# B&R Automation Studio project NAINV104C00R8L515F00 (part 8)

#### fHermesIllegalMsgNotAvlNotRdyDS.st
```iecst
(* Hermes Illegal Message - Not Available Not Ready For Downstream *)
FUNCTION fHermesIllegalMsgNotAvlNotRdyDS

	IF tyMsgType.bServiceDescription = TRUE THEN

		fHermesIllegalMsgNotAvlNotRdyDS	:= 2857;	//Receive ServiceDescription While Downstream In Not Available Not Ready State

	ELSIF tyMsgType.bBoardAvailable = TRUE THEN

		fHermesIllegalMsgNotAvlNotRdyDS	:= 2858;	//Receive BoardAvailable While Downstream In Not Available Not Ready State

	ELSIF tyMsgType.bRevokeBoardAvailable = TRUE THEN

		fHermesIllegalMsgNotAvlNotRdyDS	:= 2859;	//Receive RevokeBoardAvailable While Downstream In Not Available Not Ready State

	ELSIF tyMsgType.bRevokeMachineReady = TRUE THEN

		fHermesIllegalMsgNotAvlNotRdyDS	:= 2860;	//Receive RevokeMachineReady While Downstream In Not Available Not Ready State

	ELSIF tyMsgType.bStartTransport = TRUE THEN

		fHermesIllegalMsgNotAvlNotRdyDS	:= 2861;	//Receive StartTransport While Downstream In Not Available Not Ready State

	ELSIF tyMsgType.bStopTransport = TRUE THEN

		fHermesIllegalMsgNotAvlNotRdyDS	:= 2862;	//Receive StopTransport While Downstream In Not Available Not Ready State

	ELSIF tyMsgType.bTransportFinished = TRUE THEN

		fHermesIllegalMsgNotAvlNotRdyDS	:= 2863;	//Receive TransportFinished While Downstream In Not Available Not Ready State

	ELSIF tyMsgType.bBoardForecast = TRUE THEN

		fHermesIllegalMsgNotAvlNotRdyDS	:= 2864;	//Receive BoardForecast While Downstream In Not Available Not Ready State

	ELSE

		fHermesIllegalMsgNotAvlNotRdyDS	:= 0;

	END_IF

END_FUNCTION
```

#### fHermesIllegalMsgBrdAvlDS.st
```iecst
(* Hermes Illegal Message - Board Available For Downstream *)
FUNCTION fHermesIllegalMsgBrdAvlDS

	IF tyMsgType.bServiceDescription = TRUE THEN

		fHermesIllegalMsgBrdAvlDS	:= 2865;	//Receive ServiceDescription While Downstream In Board Available State

	ELSIF tyMsgType.bBoardAvailable = TRUE THEN

		fHermesIllegalMsgBrdAvlDS	:= 2866;	//Receive BoardAvailable While Downstream In Board Available State

	ELSIF tyMsgType.bRevokeBoardAvailable = TRUE THEN

		fHermesIllegalMsgBrdAvlDS	:= 2867;	//Receive RevokeBoardAvailable While Downstream In Board Available State

	ELSIF tyMsgType.bRevokeMachineReady = TRUE THEN

		fHermesIllegalMsgBrdAvlDS	:= 2868;	//Receive RevokeMachineReady While Downstream In Board Available State

	ELSIF (tyMsgType.bStartTransport = TRUE) AND (tyMsgType.bMachineReady = FALSE) THEN	//To Take Care When Machine Ready And StartTransport Receive In One Message

		fHermesIllegalMsgBrdAvlDS	:= 2869;	//Receive StartTransport While Downstream In Board Available State

	ELSIF tyMsgType.bStopTransport = TRUE THEN

		fHermesIllegalMsgBrdAvlDS	:= 2870;	//Receive StopTransport While Downstream In Board Available State

	ELSIF tyMsgType.bTransportFinished = TRUE THEN

		fHermesIllegalMsgBrdAvlDS	:= 2871;	//Receive TransportFinished While Downstream In Board Available State

	ELSIF tyMsgType.bBoardForecast = TRUE THEN

		fHermesIllegalMsgBrdAvlDS	:= 2872;	//Receive BoardForecast While Downstream In Board Available State

	ELSE

		fHermesIllegalMsgBrdAvlDS	:= 0;

	END_IF

END_FUNCTION
```

#### fHermesIllegalMsgMcRdyDS.st
```iecst
(* Hermes Illegal Message - Machine Ready For Downstream *)
FUNCTION fHermesIllegalMsgMcRdyDS

	IF tyMsgType.bServiceDescription = TRUE THEN

		fHermesIllegalMsgMcRdyDS	:= 2873;	//Receive ServiceDescription While Downstream In Machine Ready State

	ELSIF tyMsgType.bBoardAvailable = TRUE THEN

		fHermesIllegalMsgMcRdyDS	:= 2874;	//Receive BoardAvailable While Downstream In Machine Ready State

	ELSIF tyMsgType.bRevokeBoardAvailable = TRUE THEN

		fHermesIllegalMsgMcRdyDS	:= 2875;	//Receive RevokeBoardAvailable While Downstream In Machine Ready State

	ELSIF tyMsgType.bMachineReady = TRUE THEN

		fHermesIllegalMsgMcRdyDS	:= 2876;	//Receive MachineReady While Downstream In Machine Ready State

	ELSIF tyMsgType.bStopTransport = TRUE THEN

		fHermesIllegalMsgMcRdyDS	:= 2877;	//Receive StopTransport While Downstream In Machine Ready State

	ELSIF tyMsgType.bTransportFinished = TRUE THEN

		fHermesIllegalMsgMcRdyDS	:= 2878;	//Receive TransportFinished While Downstream In Machine Ready State

	ELSIF tyMsgType.bBoardForecast = TRUE THEN

		fHermesIllegalMsgMcRdyDS	:= 2879;	//Receive BoardForecast While Downstream In Machine Ready State

	ELSE

		fHermesIllegalMsgMcRdyDS	:= 0;

	END_IF

END_FUNCTION
```

#### fHermesIllegalMsgAvlAndRdyDS.st
```iecst
(* Hermes Illegal Message - Available And Ready For Downstream *)
FUNCTION fHermesIllegalMsgAvlAndRdyDS

	IF tyMsgType.bServiceDescription = TRUE THEN

		fHermesIllegalMsgAvlAndRdyDS	:= 2880;	//Receive ServiceDescription While Downstream In Available And Ready State

	ELSIF tyMsgType.bBoardAvailable = TRUE THEN

		fHermesIllegalMsgAvlAndRdyDS	:= 2881;	//Receive BoardAvailable While Downstream In Available And Ready State

	ELSIF tyMsgType.bRevokeBoardAvailable = TRUE THEN

		fHermesIllegalMsgAvlAndRdyDS	:= 2882;	//Receive RevokeBoardAvailable While Downstream In Available And Ready State

	ELSIF tyMsgType.bMachineReady = TRUE THEN

		fHermesIllegalMsgAvlAndRdyDS	:= 2883;	//Receive MachineReady While Downstream In Available And Ready State

	ELSIF tyMsgType.bStopTransport = TRUE THEN

		fHermesIllegalMsgAvlAndRdyDS	:= 2884;	//Receive StopTransport While Downstream In Available And Ready State

	ELSIF tyMsgType.bTransportFinished = TRUE THEN

		fHermesIllegalMsgAvlAndRdyDS	:= 2885;	//Receive TransportFinished While Downstream In Available And Ready State

	ELSIF tyMsgType.bBoardForecast = TRUE THEN

		fHermesIllegalMsgAvlAndRdyDS	:= 2886;	//Receive BoardForecast While Downstream In Available And Ready State

	ELSE

		fHermesIllegalMsgAvlAndRdyDS	:= 0;

	END_IF

END_FUNCTION
```

#### fHermesIllegalMsgTransportingDS.st
```iecst
(* Hermes Illegal Message - Transporting For Downstream *)
FUNCTION fHermesIllegalMsgTransportingDS

	IF tyMsgType.bServiceDescription = TRUE THEN

		fHermesIllegalMsgTransportingDS	:= 2887;	//Receive ServiceDescription While Downstream In Transporting State

	ELSIF tyMsgType.bBoardAvailable = TRUE THEN

		fHermesIllegalMsgTransportingDS	:= 2888;	//Receive BoardAvailable While Downstream In Transporting State

	ELSIF tyMsgType.bRevokeBoardAvailable = TRUE THEN

		fHermesIllegalMsgTransportingDS	:= 2889;	//Receive RevokeBoardAvailable While Downstream In Transporting State

	ELSIF tyMsgType.bMachineReady = TRUE THEN

		fHermesIllegalMsgTransportingDS	:= 2890;	//Receive MachineReady While Downstream In Transporting State

	ELSIF tyMsgType.bRevokeMachineReady = TRUE THEN

		fHermesIllegalMsgTransportingDS	:= 2891;	//Receive RevokeMachineReady While Downstream In Transporting State

	ELSIF tyMsgType.bStartTransport = TRUE THEN

		fHermesIllegalMsgTransportingDS	:= 2892;	//Receive StartTransport While Downstream In Transporting State

	ELSIF tyMsgType.bTransportFinished = TRUE THEN

		fHermesIllegalMsgTransportingDS	:= 2893;	//Receive TransportFinished While Downstream In Transporting State

	ELSIF tyMsgType.bBoardForecast = TRUE THEN

		fHermesIllegalMsgTransportingDS	:= 2894;	//Receive BoardForecast While Downstream In Transporting State

	ELSE

		fHermesIllegalMsgTransportingDS	:= 0;

	END_IF

END_FUNCTION
```

#### fHermesIllegalMsgTransportFiniDS.st
```iecst
(* Hermes Illegal Message - Transport Finished For Downstream *)
FUNCTION fHermesIllegalMsgTransportFiniDS

	IF tyMsgType.bServiceDescription = TRUE THEN

		fHermesIllegalMsgTransportFiniDS	:= 2895;	//Receive ServiceDescription While In Transport Finished State

	ELSIF tyMsgType.bBoardAvailable = TRUE THEN

		fHermesIllegalMsgTransportFiniDS	:= 2896;	//Receive BoardAvailable While In Transport Finished State

	ELSIF tyMsgType.bRevokeBoardAvailable = TRUE THEN

		fHermesIllegalMsgTransportFiniDS	:= 2897;	//Receive RevokeBoardAvailable While In Transport Finished State

	ELSIF tyMsgType.bMachineReady = TRUE THEN

		fHermesIllegalMsgTransportFiniDS	:= 2898;	//Receive MachineReady While In Transport Finished State

	ELSIF tyMsgType.bRevokeMachineReady = TRUE THEN

		fHermesIllegalMsgTransportFiniDS	:= 2899;	//Receive RevokeMachineReady While In Transport Finished State

	ELSIF tyMsgType.bStartTransport = TRUE THEN

		fHermesIllegalMsgTransportFiniDS	:= 2900;	//Receive StartTransport While In Transport Finished State

	ELSIF tyMsgType.bTransportFinished = TRUE THEN

		fHermesIllegalMsgTransportFiniDS	:= 2901;	//Receive TransportFinished While In Transport Finished State

	ELSIF tyMsgType.bBoardForecast = TRUE THEN

		fHermesIllegalMsgTransportFiniDS	:= 2902;	//Receive BoardForecast While In Transport Finished State

	ELSE

		fHermesIllegalMsgTransportFiniDS	:= 0;

	END_IF

END_FUNCTION
```

#### fHermesIllegalMsgTransportStopDS.st
```iecst
(* Hermes Illegal Message - Transport Stopped For Downstream *)
FUNCTION fHermesIllegalMsgTransportStopDS

	IF tyMsgType.bServiceDescription = TRUE THEN

		fHermesIllegalMsgTransportStopDS	:= 2903;	//Receive ServiceDescription While Downstream In Transport Stopped State

	ELSIF tyMsgType.bBoardAvailable = TRUE THEN

		fHermesIllegalMsgTransportStopDS	:= 2904;	//Receive BoardAvailable While Downstream In Transport Stopped State

	ELSIF tyMsgType.bRevokeBoardAvailable = TRUE THEN

		fHermesIllegalMsgTransportStopDS	:= 2905;	//Receive RevokeBoardAvailable While Downstream In Transport Stopped State

	ELSIF tyMsgType.bMachineReady = TRUE THEN

		fHermesIllegalMsgTransportStopDS	:= 2906;	//Receive MachineReady While Downstream In Transport Stopped State

	ELSIF tyMsgType.bRevokeMachineReady = TRUE THEN

		fHermesIllegalMsgTransportStopDS	:= 2907;	//Receive RevokeMachineReady While Downstream In Transport Stopped State

	ELSIF tyMsgType.bStartTransport = TRUE THEN

		fHermesIllegalMsgTransportStopDS	:= 2908;	//Receive StartTransport While Downstream In Transport Stopped State

	ELSIF tyMsgType.bStopTransport = TRUE THEN

		fHermesIllegalMsgTransportStopDS	:= 2909;	//Receive StopTransport While Downstream In Transport Stopped State

	ELSIF tyMsgType.bTransportFinished = TRUE THEN

		fHermesIllegalMsgTransportStopDS	:= 2910;	//Receive TransportFinished While Downstream In Transport Stopped State

	ELSIF tyMsgType.bBoardForecast = TRUE THEN

		fHermesIllegalMsgTransportStopDS	:= 2911;	//Receive BoardForecast While Downstream In Transport Stopped State

	ELSE

		fHermesIllegalMsgTransportStopDS	:= 0;

	END_IF

END_FUNCTION
```

#### fHermesIllegalMsgNotConnectedSvy.st
```iecst
(* Hermes Illegal Message - Not Connected For Supervisory *)
FUNCTION fHermesIllegalMsgNotConnectedSvy

	IF tyMsgType.bSetConfiguration = TRUE THEN

		fHermesIllegalMsgNotConnectedSvy	:= 2940;	//Receive SetConfiguration While Supervisory In Not Connected State

	ELSIF tyMsgType.bGetConfiguration = TRUE THEN

		fHermesIllegalMsgNotConnectedSvy	:= 2941;	//Receive GetConfiguration While Supervisory In Not Connected State

	ELSIF tyMsgType.bCurrentConfiguration = TRUE THEN

		fHermesIllegalMsgNotConnectedSvy	:= 2942;	//Receive CurrConfiguration While Supervisory In Not Connected State

	ELSIF tyMsgType.bSendWorkOrderInfo = TRUE THEN

		fHermesIllegalMsgNotConnectedSvy	:= 2943;	//Receive SendWorkOrderInfo While Supervisory In Not Connected State

	ELSIF tyMsgType.bQueryWorkOrderInfo = TRUE THEN

		fHermesIllegalMsgNotConnectedSvy	:= 2944;	//Receive QueryWorkOrderInfo While Supervisory In Not Connected State

	ELSIF tyMsgType.bBoardArrived = TRUE THEN

		fHermesIllegalMsgNotConnectedSvy	:= 2945;	//Receive BoardArrived While Supervisory In Not Connected State

	ELSIF tyMsgType.bBoardDeparted = TRUE THEN

		fHermesIllegalMsgNotConnectedSvy	:= 2946;	//Receive BoardDeparted While Supervisory In Not Connected State

	ELSE

		fHermesIllegalMsgNotConnectedSvy	:= 0;

	END_IF

END_FUNCTION
```

#### fHermesIllegalMsgSrvcDescripSvy.st
```iecst
(* Hermes Illegal Message - Supervisory Service Description *)
FUNCTION fHermesIllegalMsgSrvcDescripSvy

	IF tyMsgType.bSServiceDescription = TRUE THEN

		fHermesIllegalMsgSrvcDescripSvy	:= 2951;	//Receive Supervisory ServiceDescription While Supervisory In Service Description State

	ELSIF tyMsgType.bSetConfiguration = TRUE THEN

		fHermesIllegalMsgSrvcDescripSvy	:= 2952;	//Receive SetConfiguration While Supervisory In Service Description State

	ELSIF tyMsgType.bGetConfiguration = TRUE THEN

		fHermesIllegalMsgSrvcDescripSvy	:= 2953;	//Receive GetConfiguration While Supervisory In Service Description State

	ELSIF tyMsgType.bCurrentConfiguration = TRUE THEN

		fHermesIllegalMsgSrvcDescripSvy	:= 2954;	//Receive CurrConfiguration While Supervisory In Service Description State

	ELSIF tyMsgType.bSendWorkOrderInfo = TRUE THEN

		fHermesIllegalMsgSrvcDescripSvy	:= 2955;	//Receive SendWorkOrderInfo While Supervisory In Service Description State

	ELSIF tyMsgType.bQueryWorkOrderInfo = TRUE THEN

		fHermesIllegalMsgSrvcDescripSvy	:= 2956;	//Receive QueryWorkOrderInfo While Supervisory In Service Description State

	ELSIF tyMsgType.bBoardArrived = TRUE THEN

		fHermesIllegalMsgSrvcDescripSvy	:= 2957;	//Receive BoardArrived While Supervisory In Service Description State

	ELSIF tyMsgType.bBoardDeparted = TRUE THEN

		fHermesIllegalMsgSrvcDescripSvy	:= 2958;	//Receive BoardDeparted While Supervisory In Service Description State

	ELSE

		fHermesIllegalMsgSrvcDescripSvy	:= 0;

	END_IF

END_FUNCTION
```

#### fHermesIllegalMsgConnectedSvy.st
```iecst
(* Hermes Illegal Message - Connected For Supervisory *)
FUNCTION fHermesIllegalMsgConnectedSvy

	IF tyMsgType.bServiceDescription = TRUE THEN

		fHermesIllegalMsgConnectedSvy	:= 2963;	//Receive Supervisory ServiceDescription While Supervisory In Connected State

	ELSIF tyMsgType.bCurrentConfiguration = TRUE THEN

		fHermesIllegalMsgConnectedSvy	:= 2964;	//Receive CurrConfiguration While Supervisory In Connected State

	ELSIF tyMsgType.bQueryWorkOrderInfo = TRUE THEN

		fHermesIllegalMsgConnectedSvy	:= 2965;	//Receive QueryWorkOrderInfo While Supervisory In Connected State

	ELSIF tyMsgType.bBoardArrived = TRUE THEN

		fHermesIllegalMsgConnectedSvy	:= 2966;	//Receive BoardArrived While Supervisory In Connected State

	ELSIF tyMsgType.bBoardDeparted = TRUE THEN

		fHermesIllegalMsgConnectedSvy	:= 2967;	//Receive BoardDeparted While Supervisory In Connected State

	ELSE

		fHermesIllegalMsgConnectedSvy	:= 0;

	END_IF

END_FUNCTION
```

#### fHermesGenerateUUID.st
```iecst
(* Hermes Generate UUID *)
FUNCTION fHermesGenerateUUID

	fHermesGenerateUUID	:= TRUE;

	memset(ADR(p_sUUID) , 0 , SIZEOF(p_sUUID));

	//Year Difference: From 1970
	fConvertUSINTToHex(ADR(sTemp2) , UINT_TO_USINT((tyDTStructure.year - 1970)));
	p_sUUID	:= sTemp2;

	//Month
	fConvertUSINTToHex(ADR(sTemp2) , tyDTStructure.month);
	memcpy(ADR(p_sUUID) + LEN(p_sUUID) , ADR(sTemp2) , 2);

	//Day
	fConvertUSINTToHex(ADR(sTemp2) , tyDTStructure.day);
	memcpy(ADR(p_sUUID) + LEN(p_sUUID) , ADR(sTemp2) , 2);

	//Hour
	fConvertUSINTToHex(ADR(sTemp2) , tyDTStructure.hour);
	memcpy(ADR(p_sUUID) + LEN(p_sUUID) , ADR(sTemp2) , 2);
	memcpy(ADR(p_sUUID) + LEN(p_sUUID) , ADR('-') , 1);

	//Minute
	fConvertUSINTToHex(ADR(sTemp2) , tyDTStructure.minute);
	memcpy(ADR(p_sUUID) + LEN(p_sUUID) , ADR(sTemp2) , 2);

	//Second
	fConvertUSINTToHex(ADR(sTemp2) , tyDTStructure.second);
	memcpy(ADR(p_sUUID) + LEN(p_sUUID) , ADR(sTemp2) , 2);
	memcpy(ADR(p_sUUID) + LEN(p_sUUID) , ADR('-') , 1);

	//Millisec
	fConvertUINTToHex(ADR(sTemp4) , tyDTStructure.millisec);
	memcpy(ADR(p_sUUID) + LEN(p_sUUID) , ADR(sTemp4) , 4);
	memcpy(ADR(p_sUUID) + LEN(p_sUUID) , ADR('-') , 1);

	//Microsec
	fConvertUINTToHex(ADR(sTemp4) , tyDTStructure.microsec);
	memcpy(ADR(p_sUUID) + LEN(p_sUUID) , ADR(sTemp4) , 4);
	memcpy(ADR(p_sUUID) + LEN(p_sUUID) , ADR('-') , 1);

	//Mac Address
	fConvertUSINTToHex(ADR(sTemp2) , a_usiMacAddr[0]);
	memcpy(ADR(p_sUUID) + LEN(p_sUUID) , ADR(sTemp2) , 2);

	fConvertUSINTToHex(ADR(sTemp2) , a_usiMacAddr[1]);
	memcpy(ADR(p_sUUID) + LEN(p_sUUID) , ADR(sTemp2) , 2);

	fConvertUSINTToHex(ADR(sTemp2) , a_usiMacAddr[2]);
	memcpy(ADR(p_sUUID) + LEN(p_sUUID) , ADR(sTemp2) , 2);

	fConvertUSINTToHex(ADR(sTemp2) , a_usiMacAddr[3]);
	memcpy(ADR(p_sUUID) + LEN(p_sUUID) , ADR(sTemp2) , 2);

	fConvertUSINTToHex(ADR(sTemp2) , a_usiMacAddr[4]);
	memcpy(ADR(p_sUUID) + LEN(p_sUUID) , ADR(sTemp2) , 2);

	fConvertUSINTToHex(ADR(sTemp2) , a_usiMacAddr[5]);
	memcpy(ADR(p_sUUID) + LEN(p_sUUID) , ADR(sTemp2) , 2);

END_FUNCTION
```

#### fHermesGetTimestamp.st
```iecst
(* Hermes Get Timestamp *)
FUNCTION fHermesGetTimestamp

	fHermesGetTimestamp	:= TRUE;

	memset(ADR(p_sTimestamp) , 0 , SIZEOF(p_sTimestamp));
	memset(ADR(sYear) , 0 , SIZEOF(sYear));
	memset(ADR(sMonth) , 0 , SIZEOF(sMonth));
	memset(ADR(sDay) , 0 , SIZEOF(sDay));
	memset(ADR(sHour) , 0 , SIZEOF(sHour));
	memset(ADR(sMinute) , 0 , SIZEOF(sMinute));
	memset(ADR(sSecond) , 0 , SIZEOF(sSecond));
	memset(ADR(sMillisec) , 0 , SIZEOF(sMillisec));

	sYear	:= UINT_TO_STRING(tyDTStructure.year);

	IF tyDTStructure.year < 10 THEN
		memcpy(ADR(sYear) + 3 , ADR(sYear) , 1);
		memcpy(ADR(sYear) , ADR('000') , 3);
	ELSIF tyDTStructure.year < 100 THEN
		memcpy(ADR(sYear) + 2 , ADR(sYear) , 2);
		memcpy(ADR(sYear) , ADR('000') , 2);
	ELSIF tyDTStructure.year < 1000 THEN
		memcpy(ADR(sYear) + 1 , ADR(sYear) , 3);
		memcpy(ADR(sYear) , ADR('000') , 1);
	END_IF

	sMonth	:= USINT_TO_STRING(tyDTStructure.month);

	IF tyDTStructure.month < 10 THEN
		memcpy(ADR(sMonth) + 1 , ADR(sMonth) , 1);
		memcpy(ADR(sMonth) , ADR('0') , 1);
	END_IF

	sDay	:= USINT_TO_STRING(tyDTStructure.day);

	IF tyDTStructure.day < 10 THEN
		memcpy(ADR(sDay) + 1 , ADR(sDay) , 1);
		memcpy(ADR(sDay) , ADR('0') , 1);
	END_IF

	sHour	:= USINT_TO_STRING(tyDTStructure.hour);

	IF tyDTStructure.hour < 10 THEN
		memcpy(ADR(sHour) + 1 , ADR(sHour) , 1);
		memcpy(ADR(sHour) , ADR('0') , 1);
	END_IF

	sMinute	:= USINT_TO_STRING(tyDTStructure.minute);

	IF tyDTStructure.minute < 10 THEN
		memcpy(ADR(sMinute) + 1 , ADR(sMinute) , 1);
		memcpy(ADR(sMinute) , ADR('0') , 1);
	END_IF

	sSecond	:= USINT_TO_STRING(tyDTStructure.second);

	IF tyDTStructure.second < 10 THEN
		memcpy(ADR(sSecond) + 1 , ADR(sSecond) , 1);
		memcpy(ADR(sSecond) , ADR('0') , 1);
	END_IF

	sMillisec	:= UINT_TO_STRING(tyDTStructure.millisec);

	memcpy(ADR(p_sTimestamp) + LEN(p_sTimestamp) , ADR(sYear) , 4);
	memcpy(ADR(p_sTimestamp) + LEN(p_sTimestamp) , ADR('-') , 1);
	memcpy(ADR(p_sTimestamp) + LEN(p_sTimestamp) , ADR(sMonth) , 2);
	memcpy(ADR(p_sTimestamp) + LEN(p_sTimestamp) , ADR('-') , 1);
	memcpy(ADR(p_sTimestamp) + LEN(p_sTimestamp) , ADR(sDay) , 2);
	memcpy(ADR(p_sTimestamp) + LEN(p_sTimestamp) , ADR('T') , 1);
	memcpy(ADR(p_sTimestamp) + LEN(p_sTimestamp) , ADR(sHour) , 2);
	memcpy(ADR(p_sTimestamp) + LEN(p_sTimestamp) , ADR(':') , 1);
	memcpy(ADR(p_sTimestamp) + LEN(p_sTimestamp) , ADR(sMinute) , 2);
	memcpy(ADR(p_sTimestamp) + LEN(p_sTimestamp) , ADR(':') , 1);
	memcpy(ADR(p_sTimestamp) + LEN(p_sTimestamp) , ADR(sSecond) , 2);
	memcpy(ADR(p_sTimestamp) + LEN(p_sTimestamp) , ADR('.') , 1);
	memcpy(ADR(p_sTimestamp) + LEN(p_sTimestamp) , ADR(sMillisec) , LEN(sMillisec));

END_FUNCTION
```

#### fHermesRmvOneMsgSend.st
```iecst
(* Hermes Remove One Message Send Buffer *)
FUNCTION fHermesRmvOneMsgSend

	fHermesRmvOneMsgSend	:= TRUE;

	memcpy(ADR(pa_eMsgSend[0]) , ADR(pa_eMsgSend[1]) , SIZEOF(pa_eMsgSend[0]) * 50);
	pa_eMsgSend[50]	:= HermesMsgTypeNA;
	p_udiIdx		:= p_udiIdx - 1;

END_FUNCTION
```

#### fHermesAddOneMsgSend.st
```iecst
(* Hermes Add One Message Send Buffer *)
FUNCTION fHermesAddOneMsgSend

	fHermesAddOneMsgSend	:= TRUE;

	pa_eMsgSend[p_udiIdx]	:= eMsgType;
	p_udiIdx				:= p_udiIdx + 1;

END_FUNCTION
```

#### fHermesRmvOneCmdTyp.st
```iecst
(* Hermes Remove One Message Send Buffer *)
FUNCTION fHermesRmvOneCmdTyp

	fHermesRmvOneCmdTyp	:= TRUE;

	memcpy(ADR(pa_eCmd[0]) , ADR(pa_eCmd[1]) , SIZEOF(pa_eCmd[0]) * 10);
	pa_eCmd[10]	:= HermesCommandUndefined;
	p_udiIdx		:= p_udiIdx - 1;

END_FUNCTION
```

#### fHermesAddOneCmdTyp.st
```iecst
(* Hermes Add One Message Send Buffer *)
FUNCTION fHermesAddOneCmdTyp

	fHermesAddOneCmdTyp	:= TRUE;

	pa_eCmd[p_udiIdx]		:= eCmd;
	p_udiIdx				:= p_udiIdx + 1;

END_FUNCTION
```

#### fHermesChkParamCommand.st
```iecst
(* Hermes Checking Parameter SendWorkOrderId & QueryWorkOrderId *)
FUNCTION fHermesChkParamCommand

	fHermesChkParamCommand	:= 0;

	IF tyCommand.tyAvl.bCommand = TRUE THEN
		//(tyCommand.tyData.eCommand < 0 OR tyCommand.tyData.eCommand > 9999)
		IF tyCommand.tyData.eCommand < 0 OR tyCommand.tyData.eCommand > 9999  THEN

			fHermesChkParamCommand	:= 8888;	//Command not supported

		END_IF

	ELSE

		fHermesChkParamCommand	:= 7777;	//Command Message missing Attribute Command

	END_IF

END_FUNCTION
```

#### fHermesAddOneCommandGate.st
```iecst
(* Hermes Checking Parameter SendWorkOrderId & QueryWorkOrderId *)
FUNCTION fHermesAddOneCommandGate

	fHermesAddOneCommandGate	:= p_udiIdx;
	tyCommandProcessList[p_udiIdx].bUSTrueDSFalse :=  bUsTrueDsFalse;
	tyCommandProcessList[p_udiIdx].udiCommandParam :=  ADR(tyHermesCmdParam);
	tyCommandProcessList[p_udiIdx].udiComMode := ADR(udiComMode) ;
	tyCommandProcessList[p_udiIdx].udiInterfaceString :=  ADR(sInterface);
	p_udiIdx := p_udiIdx +1;
END_FUNCTION
```

#### fHermesBoardCastCommand.st
```iecst
(* Hermes BroadCast Command To other interface *)
FUNCTION fHermesBroadCastCommand

END_FUNCTION
```

#### fbHermesProcessCmd.st
```iecst
(* ProcessCmd *)
FUNCTION fHermesProcessCmd

	FOR usiIdx  := 0 TO SIZEOF(tyCommandProcessList)/SIZEOF(tyCommandProcessList[0]) DO
		IF tyCommandProcessList[usiIdx].udiCommandParam <> 0 AND tyCommandProcessList[usiIdx].udiComMode <> 0 AND tyCommandProcessList[usiIdx].udiInterfaceString <> 0 THEN
			p_tyHermesCmdParam ACCESS tyCommandProcessList[usiIdx].udiCommandParam;
			p_tyHermesCmdPause ACCESS ADR(tyHermesCmdPause[usiIdx]);

			//------- Process Rcv and BoardCast if not suppported ------//
			IF p_tyHermesCmdParam.usiCommandIdx <> a_usiCommandIdx[usiIdx] THEN //track command idx
				//Checking Processability and feature
				usiPrevCmdIdx := a_usiCommandIdx[usiIdx];

				//Rcv
				IF p_tyHermesCmdPause.bFeatureRequestTo THEN
					fHermesRcvCmdReqToPause(ADR(a_usiCommandIdx[usiIdx]),ADR(p_tyHermesCmdParam),ADR(p_tyHermesCmdPause));
				END_IF

				IF  p_tyHermesCmdPause.bFeatureRequestFrom THEN
					fHermesRcvCmdReqFromPause(ADR(a_usiCommandIdx[usiIdx]),ADR(p_tyHermesCmdParam),ADR(p_tyHermesCmdPause))	;
				END_IF

				//Adding Command to other interface if not able to execute, Polling
				IF usiPrevCmdIdx <> a_usiCommandIdx[usiIdx] THEN 	//if not supported, then broadcast
					FOR usiCmpIdx  := 0 TO SIZEOF(tyCommandProcessList)/SIZEOF(tyCommandProcessList[0]) DO //loop other
						IF usiIdx <> usiCmpIdx  THEN //not self
							p_sCmpInterface ACCESS tyCommandProcessList[usiCmpIdx].udiCommandParam;
							p_udiComMode ACCESS tyCommandProcessList[usiCmpIdx].udiComMode;
							IF p_sInterface <> p_sCmpInterface AND p_udiComMode = 0 THEN //not same interfafce and is Hermes Communication
								p_udiHermesCmpCmdParam ACCESS tyCommandProcessList[usiCmpIdx].udiCommandParam;
								fHermesAddOneCmdTyp(ADR(p_udiHermesCmpCmdParam.a_eCommandSndQ),ADR(p_udiHermesCmpCmdParam.udiMsgCmdBffr),p_tyHermesCmdParam.eCommand);
							END_IF
						END_IF
					END_FOR
				END_IF
			END_IF

				//------- Process Send if supported  ------//
			IF p_tyHermesCmdPause.bFeatureRequestTo THEN
				fHermesSndCmdReqToPause(ADR(p_tyHermesCmdParam),ADR(p_tyHermesCmdPause));
			END_IF

			IF  p_tyHermesCmdPause.bFeatureRequestFrom THEN
				fHermesSndCmdReqFromPause(ADR(p_tyHermesCmdParam),ADR(p_tyHermesCmdPause));
			END_IF

		END_IF
	END_FOR

END_FUNCTION
```

#### fHermesRcvCmdReqFromPause.st
```iecst
(* ProcessCmd *)
FUNCTION fHermesRcvCmdReqFromPause

	IF	p_tyHermesCmdParam.eCommand = HermesCommandRequestPause THEN
			p_tyHermesCmdPause.bUnlockCoverSigFrom := TRUE ;
			p_usiCommandIdx := p_usiCommandIdx +1 ;
	ELSIF p_tyHermesCmdParam.eCommand = HermesCommandResumeOperation THEN
			p_tyHermesCmdPause.bUnlockCoverSigFrom := FALSE;
			p_usiCommandIdx := p_usiCommandIdx +1 ;
	END_IF

END_FUNCTION
```

#### fHermesRcvCmdReqToPause.st
```iecst
(* ProcessCmd *)
FUNCTION fHermesRcvCmdReqToPause

	IF p_tyHermesCmdParam.eCommand = HermesCommandConfirmPause THEN
		p_tyHermesCmdPause.bMachineSafetySigFrom := TRUE;
		p_usiCommandIdx := p_usiCommandIdx +1 ;
	END_IF

END_FUNCTION
```

#### fHermesRcvCmdReqFromLockCov.st
```iecst
(* ProcessCmd *)
FUNCTION fHermesRcvCmdReqFromLockCov

	IF	p_tyHermesCmdParam.eCommand = HermesCommandLockInputConveyor THEN
			p_tyHermesCmdLockCov.bOvenInfoFrom := TRUE ;
			p_usiCommandIdx := p_usiCommandIdx +1 ;
	ELSIF p_tyHermesCmdParam.eCommand = HermesCommandUnLockInputConveyor THEN
			p_tyHermesCmdLockCov.bOvenInfoFrom := FALSE;
			p_usiCommandIdx := p_usiCommandIdx +1 ;
	END_IF

END_FUNCTION
```

#### fHermesRcvCmdReqFromOvenInfeed.st
```iecst
(* ProcessCmd *)
FUNCTION fHermesRcvCmdReqFromOvenInfeed

	IF	p_tyHermesCmdParam.eCommand = HermesCommandOvenInfeed THEN
			p_tyHermesCmdOvenInfeed.bOvenInfeedFrom := TRUE ;
			p_usiCommandIdx := p_usiCommandIdx +1 ;
	ELSIF p_tyHermesCmdParam.eCommand = HermesCommandOvenInfeed THEN
			p_tyHermesCmdOvenInfeed.bOvenInfeedFrom := FALSE;
			p_usiCommandIdx := p_usiCommandIdx +1 ;
	END_IF

END_FUNCTION
```

#### fHermesSndCmdReqFromPause.st
```iecst
(* ProcessCmd *)
FUNCTION fHermesSndCmdReqFromPause

	IF p_tyHermesCmdPause.bMachineSafetySigTo <> p_tyHermesCmdPause.bPrevMachineSafetySigTo THEN
		IF p_tyHermesCmdPause.bMachineSafetySigTo = TRUE THEN
			fHermesAddOneCmdTyp(ADR(p_tyHermesCmdParam.a_eCommandSndQ),ADR(p_tyHermesCmdParam.udiMsgCmdBffr),HermesCommandConfirmPause);
		END_IF
		p_tyHermesCmdPause.bPrevMachineSafetySigTo := p_tyHermesCmdPause.bMachineSafetySigTo;
	END_IF

END_FUNCTION
```

#### fHermesSndCmdReqToPause.st
```iecst
(* ProcessCmd *)
FUNCTION fHermesSndCmdReqToPause

	IF p_tyHermesCmdPause.bUnlockCoverSigTo <> p_tyHermesCmdPause.bPrevUnlockCoverSigTo THEN
		IF p_tyHermesCmdPause.bUnlockCoverSigTo = TRUE THEN
			fHermesAddOneCmdTyp(ADR(p_tyHermesCmdParam.a_eCommandSndQ),ADR(p_tyHermesCmdParam.udiMsgCmdBffr),HermesCommandRequestPause);
		ELSE
			fHermesAddOneCmdTyp(ADR(p_tyHermesCmdParam.a_eCommandSndQ),ADR(p_tyHermesCmdParam.udiMsgCmdBffr),HermesCommandResumeOperation);
			p_tyHermesCmdPause.bMachineSafetySigFrom := FALSE;
		END_IF
		p_tyHermesCmdPause.bPrevUnlockCoverSigTo := p_tyHermesCmdPause.bUnlockCoverSigTo;
	END_IF

END_FUNCTION
```

#### fHermesSndCmdReqToLockConv.st
```iecst
(* ProcessCmd *)
FUNCTION fHermesSndCmdReqToLockConv

	IF p_tyHermesCmdLockCov.bOvenInfoTo <> p_tyHermesCmdLockCov.bPrevOvenInfoTo THEN
		IF p_tyHermesCmdLockCov.bOvenInfoTo = TRUE THEN
			fHermesAddOneCmdTyp(ADR(p_tyHermesCmdParam.a_eCommandSndQ),ADR(p_tyHermesCmdParam.udiMsgCmdBffr),HermesCommandLockInputConveyor);
		ELSE
			fHermesAddOneCmdTyp(ADR(p_tyHermesCmdParam.a_eCommandSndQ),ADR(p_tyHermesCmdParam.udiMsgCmdBffr),HermesCommandUnLockInputConveyor);
		END_IF
		p_tyHermesCmdLockCov.bPrevOvenInfoTo := p_tyHermesCmdLockCov.bOvenInfoTo;
	END_IF

END_FUNCTION
```

#### fHermesSndCmdReqToOvenInfeed.st
```iecst
(* ProcessCmd *)
FUNCTION fHermesSndCmdReqToOvenInfeed

	IF p_tyHermesCmdOvenInfeed.bOvenInfeedTo <> p_tyHermesCmdOvenInfeed.bFeatureOvenInfeedFrom THEN
		IF p_tyHermesCmdOvenInfeed.bOvenInfeedTo = TRUE THEN
			fHermesAddOneCmdTyp(ADR(p_tyHermesCmdParam.a_eCommandSndQ),ADR(p_tyHermesCmdParam.udiMsgCmdBffr),HermesCommandOvenInfeed);
		ELSE
			fHermesAddOneCmdTyp(ADR(p_tyHermesCmdParam.a_eCommandSndQ),ADR(p_tyHermesCmdParam.udiMsgCmdBffr),HermesCommandOvenInfeed);
		END_IF
		p_tyHermesCmdOvenInfeed.bPrevOvenInfeedTo := p_tyHermesCmdOvenInfeed.bOvenInfeedTo;
	END_IF

END_FUNCTION
```

#### fHermesBrdAvltoBF.st
```iecst
(* Hermes Add One Message Send Buffer *)
FUNCTION fHermesBrdAvltoBF

	fHermesBrdAvltoBF := 0;

	tyHermesBoardForecast.tyData.sBoardId := tyHermesBoardAvailable.tyData.sBoardId;
	tyHermesBoardForecast.tyData.sBoardIdCreatedBy := tyHermesBoardAvailable.tyData.sBoardIdCreatedBy;
	tyHermesBoardForecast.tyData.eFailedBoard := tyHermesBoardAvailable.tyData.eFailedBoard;
	tyHermesBoardForecast.tyData.sProductTypeId := tyHermesBoardAvailable.tyData.sProductTypeId;
	tyHermesBoardForecast.tyData.eFlippedBoard := tyHermesBoardAvailable.tyData.eFlippedBoard ;
	tyHermesBoardForecast.tyData.sTopBarcode := 	tyHermesBoardAvailable.tyData.sTopBarcode;
	tyHermesBoardForecast.tyData.sBottomBarcode := 	tyHermesBoardAvailable.tyData.sBottomBarcode ;
	tyHermesBoardForecast.tyData.rLength	:= 	tyHermesBoardAvailable.tyData.rLength;
	tyHermesBoardForecast.tyData.rWidth	:= 	tyHermesBoardAvailable.tyData.rWidth;
	tyHermesBoardForecast.tyData.rThickness := 	tyHermesBoardAvailable.tyData.rThickness;
	tyHermesBoardForecast.tyData.rConveyorSpeed := 	tyHermesBoardAvailable.tyData.rConveyorSpeed;
	tyHermesBoardForecast.tyData.rTopClearanceHeight := 	tyHermesBoardAvailable.tyData.rTopClearanceHeight;
	tyHermesBoardForecast.tyData.rBottomClearanceHeight := 	tyHermesBoardAvailable.tyData.rBottomClearanceHeight;
	tyHermesBoardForecast.tyData.rWeight := 	tyHermesBoardAvailable.tyData.rWeight;
	tyHermesBoardForecast.tyData.sWorkOrderId := 	tyHermesBoardAvailable.tyData.sWorkOrderId;
	tyHermesBoardForecast.tyData.sBatchId := 	tyHermesBoardAvailable.tyData.sBatchId;

	tyHermesBoardForecast.tyAvl.bBoardId := tyHermesBoardAvailable.tyData.sBoardId <> '';
	tyHermesBoardForecast.tyAvl.bBoardIdCreatedBy := tyHermesBoardAvailable.tyData.sBoardIdCreatedBy <> '';
	tyHermesBoardForecast.tyAvl.bFailedBoard := TRUE;// tyHermesBoardAvailable.tyData.eFailedBoard <> 0;
	tyHermesBoardForecast.tyAvl.bProductTypeId := tyHermesBoardAvailable.tyData.sProductTypeId <> '';
	tyHermesBoardForecast.tyAvl.bFlippedBoard := TRUE ;//tyHermesBoardAvailable.tyData.eFlippedBoard <>0  ;
	tyHermesBoardForecast.tyAvl.bTopBarcode := 	tyHermesBoardAvailable.tyData.sTopBarcode <> '';
	tyHermesBoardForecast.tyAvl.bBottomBarcode := 	tyHermesBoardAvailable.tyData.sBottomBarcode <> '';
	tyHermesBoardForecast.tyAvl.bLength	:= 	tyHermesBoardAvailable.tyData.rLength <>0;
	tyHermesBoardForecast.tyAvl.bWidth	:= 	tyHermesBoardAvailable.tyData.rWidth <>0;
	tyHermesBoardForecast.tyAvl.bThickness := 	tyHermesBoardAvailable.tyData.rThickness <>0;
	tyHermesBoardForecast.tyAvl.bConveyorSpeed := 	tyHermesBoardAvailable.tyData.rConveyorSpeed <>0;
	tyHermesBoardForecast.tyAvl.bTopClearanceHeight := 	tyHermesBoardAvailable.tyData.rTopClearanceHeight <>0;
	tyHermesBoardForecast.tyAvl.bBottomClearanceHeight := 	tyHermesBoardAvailable.tyData.rBottomClearanceHeight<>0;
	tyHermesBoardForecast.tyAvl.bWeight := 	tyHermesBoardAvailable.tyData.rWeight<>0;
	tyHermesBoardForecast.tyAvl.bWorkOrderId := 	tyHermesBoardAvailable.tyData.sWorkOrderId <> '';
	tyHermesBoardForecast.tyAvl.bBatchId := 	tyHermesBoardAvailable.tyData.sBatchId <> '';

END_FUNCTION
```

#### fHermesAddEditAttribBrdAvlDat.st - not listed in the package file held
```iecst
(* Hermes Add Edit Attribute Value to BrvAvlDat *)
FUNCTION fHermesAddEditAttribBrdAvlDat

	fHermesAddEditAttribBrdAvlDat := 0;
	fConvertToLower_254(ADR(sTitleLowerCase) , sAttributeTiltle);

	FOR i := 0 TO 200 DO //search for the board action and update / add if not exist
		IF (p_tyHermesBrdAvlDat.a_tyXMLTableDataBrdAvl[i].sTitle = 'AT') THEN
			fConvertToLower_254(ADR(sLowerCase) , p_tyHermesBrdAvlDat.a_tyXMLTableDataBrdAvl[i].sValue);
			IF (sLowerCase = sTitleLowerCase) THEN
				IF p_tyHermesBrdAvlDat.a_tyXMLTableDataBrdAvl[i+1].sTitle = 'AV' THEN
					p_tyHermesBrdAvlDat.a_tyXMLTableDataBrdAvl[i+1].sValue	:= sAttributeValue ; //if Action already in XMLTable
					EXIT;
				END_IF
			END_IF
		ELSIF (p_tyHermesBrdAvlDat.a_tyXMLTableDataBrdAvl[i].sTitle = 'EN') AND (p_tyHermesBrdAvlDat.a_tyXMLTableDataBrdAvl[i+1].sTitle = 'ST') THEN //with subboard tag
			fConvertToLower_254(ADR(sLowerCase) , p_tyHermesBrdAvlDat.a_tyXMLTableDataBrdAvl[i+1].sValue);
			IF (sLowerCase = 'subboards') THEN
				udiHermesAttributeEndIdx := i;
			END_IF
		ELSIF (p_tyHermesBrdAvlDat.a_tyXMLTableDataBrdAvl[i].sTitle = 'ES') AND (p_tyHermesBrdAvlDat.a_tyXMLTableDataBrdAvl[i+1].sTitle = 'ET') THEN //no subboard tag
			fConvertToLower_254(ADR(sLowerCase) , p_tyHermesBrdAvlDat.a_tyXMLTableDataBrdAvl[i+1].sValue);
			IF (sLowerCase = 'hermes') THEN
				udiHermesAttributeEndIdx := i;
			END_IF
		ELSIF (p_tyHermesBrdAvlDat.a_tyXMLTableDataBrdAvl[i].sTitle = 'ET') AND (p_tyHermesBrdAvlDat.a_tyXMLTableDataBrdAvl[i+1].sTitle = 'EN') THEN //very end of Hermes tag
			fConvertToLower_254(ADR(sLowerCase) , p_tyHermesBrdAvlDat.a_tyXMLTableDataBrdAvl[i].sValue);
			IF (sLowerCase = 'hermes') THEN
				udiHermesBAEndIdx := i+1;
			END_IF
		END_IF
	END_FOR
	IF i = 201 THEN //if not found  action attibute in Hermes Message, create own Action Attribute
		memcpy(ADR(p_tyHermesBrdAvlDat.a_tyXMLTableDataBrdAvl[udiHermesAttributeEndIdx])+SIZEOF(p_tyHermesBrdAvlDat.a_tyXMLTableDataBrdAvl[0])*2,
		ADR(p_tyHermesBrdAvlDat.a_tyXMLTableDataBrdAvl[udiHermesAttributeEndIdx]),
		(udiHermesBAEndIdx - udiHermesAttributeEndIdx)*SIZEOF(p_tyHermesBrdAvlDat.a_tyXMLTableDataBrdAvl[0]));
		p_tyHermesBrdAvlDat.a_tyXMLTableDataBrdAvl[udiHermesAttributeEndIdx].sTitle := 'AT';
		p_tyHermesBrdAvlDat.a_tyXMLTableDataBrdAvl[udiHermesAttributeEndIdx].sValue := sAttributeTiltle;
		p_tyHermesBrdAvlDat.a_tyXMLTableDataBrdAvl[udiHermesAttributeEndIdx].uiSize := LEN(p_tyHermesBrdAvlDat.a_tyXMLTableDataBrdAvl[udiHermesAttributeEndIdx].sValue);
		p_tyHermesBrdAvlDat.a_tyXMLTableDataBrdAvl[udiHermesAttributeEndIdx+1].sTitle := 'AV';
		p_tyHermesBrdAvlDat.a_tyXMLTableDataBrdAvl[udiHermesAttributeEndIdx+1].sValue := sAttributeValue ;
		p_tyHermesBrdAvlDat.a_tyXMLTableDataBrdAvl[udiHermesAttributeEndIdx+1].uiSize := LEN(p_tyHermesBrdAvlDat.a_tyXMLTableDataBrdAvl[udiHermesAttributeEndIdx+1].sValue);
	END_IF

END_FUNCTION
```

#### fHermesDeleteAttribBrdAvlDat.st - not listed in the package file held
```iecst
(* Hermes Delete Attribute Value from BrvAvlDat *)
FUNCTION fHermesDeleteAttribBrdAvlDat

	fHermesDeleteAttribBrdAvlDat := 0;
	fConvertToLower_254(ADR(sTitleLowerCase) , sAttributeTiltle);
	usiBrdDatSize := SIZEOF(p_tyHermesBrdAvlDat.a_tyXMLTableDataBrdAvl)/SIZEOF(p_tyHermesBrdAvlDat.a_tyXMLTableDataBrdAvl[1]);
	FOR i := 0 TO usiBrdDatSize  DO //search for the board action and update / add if not exist
		IF (p_tyHermesBrdAvlDat.a_tyXMLTableDataBrdAvl[i].sTitle = 'AT') THEN
			fConvertToLower_254(ADR(sLowerCase) , p_tyHermesBrdAvlDat.a_tyXMLTableDataBrdAvl[i].sValue);
			IF (sLowerCase = sTitleLowerCase) THEN
				IF p_tyHermesBrdAvlDat.a_tyXMLTableDataBrdAvl[i+1].sTitle = 'AV' THEN
					//p_tyHermesBrdAvlDat.a_tyXMLTableDataBrdAvl[i+1].sValue	:= sAttributeValue ; //if Action already in XMLTable
					udiHermesAttributeEndIdx := i;
					EXIT;
				END_IF
			END_IF

		END_IF
	END_FOR
	IF i <> usiBrdDatSize THEN
		memmove(ADR(p_tyHermesBrdAvlDat.a_tyXMLTableDataBrdAvl[0])+udiHermesAttributeEndIdx*SIZEOF(p_tyHermesBrdAvlDat.a_tyXMLTableDataBrdAvl[0])
		,ADR(p_tyHermesBrdAvlDat.a_tyXMLTableDataBrdAvl[0])+(udiHermesAttributeEndIdx+2)*SIZEOF(p_tyHermesBrdAvlDat.a_tyXMLTableDataBrdAvl[0])
		,SIZEOF(p_tyHermesBrdAvlDat.a_tyXMLTableDataBrdAvl[0])*(usiBrdDatSize-(i+2)));
		fHermesDeleteAttribBrdAvlDat := TRUE;
	END_IF

END_FUNCTION
```

#### fHermesFormReplyWorkOrderInfo.st - not listed in the package file held
```iecst
(* Hermes Form Reply Work Order Info Table Data (Total Index Written In Table) *)
FUNCTION fHermesFormReplyWorkOrderInfo

	memset(ADR(pa_tyXMLTable) , 0 , SIZEOF(pa_tyXMLTable));
	iTotalIdxWrite	:= 0;

	fHermesGetTimestamp(ADR(sTimestamp) , tyDTStructure);

	pa_tyXMLTable[iTotalIdxWrite].sTitle	:= 'ST';
	pa_tyXMLTable[iTotalIdxWrite].sValue	:= 'Hermes';
	pa_tyXMLTable[iTotalIdxWrite].uiSize	:= LEN(pa_tyXMLTable[iTotalIdxWrite].sValue);

	iTotalIdxWrite	:= iTotalIdxWrite + 1;

	pa_tyXMLTable[iTotalIdxWrite].sTitle	:= 'AT';
	pa_tyXMLTable[iTotalIdxWrite].sValue	:= 'Timestamp';
	pa_tyXMLTable[iTotalIdxWrite].uiSize	:= LEN(pa_tyXMLTable[iTotalIdxWrite].sValue);

	iTotalIdxWrite	:= iTotalIdxWrite + 1;

	pa_tyXMLTable[iTotalIdxWrite].sTitle	:= 'AV';
	pa_tyXMLTable[iTotalIdxWrite].sValue	:= sTimestamp;
	pa_tyXMLTable[iTotalIdxWrite].uiSize	:= LEN(pa_tyXMLTable[iTotalIdxWrite].sValue);

	iTotalIdxWrite	:= iTotalIdxWrite + 1;

	pa_tyXMLTable[iTotalIdxWrite].sTitle	:= 'EN';
	pa_tyXMLTable[iTotalIdxWrite].sValue	:= '';
	pa_tyXMLTable[iTotalIdxWrite].uiSize	:= LEN(pa_tyXMLTable[iTotalIdxWrite].sValue);

	iTotalIdxWrite	:= iTotalIdxWrite + 1;

	pa_tyXMLTable[iTotalIdxWrite].sTitle	:= 'ST';
	pa_tyXMLTable[iTotalIdxWrite].sValue	:= 'ReplyWorkOrderInfo';
	pa_tyXMLTable[iTotalIdxWrite].uiSize	:= LEN(pa_tyXMLTable[iTotalIdxWrite].sValue);

	iTotalIdxWrite	:= iTotalIdxWrite + 1;

	IF tyParameter.tyAvl.bWorkOrderId = TRUE THEN
		pa_tyXMLTable[iTotalIdxWrite].sTitle	:= 'AT';
		pa_tyXMLTable[iTotalIdxWrite].sValue	:= 'WorkOrderId';
		pa_tyXMLTable[iTotalIdxWrite].uiSize	:= LEN(pa_tyXMLTable[iTotalIdxWrite].sValue);

		iTotalIdxWrite	:= iTotalIdxWrite + 1;

		pa_tyXMLTable[iTotalIdxWrite].sTitle	:= 'AV';
		pa_tyXMLTable[iTotalIdxWrite].sValue	:= tyParameter.tyData.sWorkOrderId;
		pa_tyXMLTable[iTotalIdxWrite].uiSize	:= LEN(pa_tyXMLTable[iTotalIdxWrite].sValue);

		iTotalIdxWrite	:= iTotalIdxWrite + 1;
	END_IF

	IF tyParameter.tyAvl.bBatchId = TRUE THEN
		pa_tyXMLTable[iTotalIdxWrite].sTitle	:= 'AT';
		pa_tyXMLTable[iTotalIdxWrite].sValue	:= 'BatchId';
		pa_tyXMLTable[iTotalIdxWrite].uiSize	:= LEN(pa_tyXMLTable[iTotalIdxWrite].sValue);

		iTotalIdxWrite	:= iTotalIdxWrite + 1;

		pa_tyXMLTable[iTotalIdxWrite].sTitle	:= 'AV';
		pa_tyXMLTable[iTotalIdxWrite].sValue	:= tyParameter.tyData.sBatchId;
		pa_tyXMLTable[iTotalIdxWrite].uiSize	:= LEN(pa_tyXMLTable[iTotalIdxWrite].sValue);

		iTotalIdxWrite	:= iTotalIdxWrite + 1;
	END_IF

	IF tyParameter.tyAvl.bStatus = TRUE THEN
		pa_tyXMLTable[iTotalIdxWrite].sTitle	:= 'AT';
		pa_tyXMLTable[iTotalIdxWrite].sValue	:= 'Status';
		pa_tyXMLTable[iTotalIdxWrite].uiSize	:= LEN(pa_tyXMLTable[iTotalIdxWrite].sValue);

		iTotalIdxWrite	:= iTotalIdxWrite + 1;

		pa_tyXMLTable[iTotalIdxWrite].sTitle	:= 'AV';
		pa_tyXMLTable[iTotalIdxWrite].sValue	:= INT_TO_STRING(tyParameter.tyData.iStatus);
		pa_tyXMLTable[iTotalIdxWrite].uiSize	:= LEN(pa_tyXMLTable[iTotalIdxWrite].sValue);

		iTotalIdxWrite	:= iTotalIdxWrite + 1;
	END_IF

	pa_tyXMLTable[iTotalIdxWrite].sTitle	:= 'ES';
	pa_tyXMLTable[iTotalIdxWrite].sValue	:= '';
	pa_tyXMLTable[iTotalIdxWrite].uiSize	:= LEN(pa_tyXMLTable[iTotalIdxWrite].sValue);

	iTotalIdxWrite	:= iTotalIdxWrite + 1;

	pa_tyXMLTable[iTotalIdxWrite].sTitle	:= 'ET';
	pa_tyXMLTable[iTotalIdxWrite].sValue	:= 'Hermes';
	pa_tyXMLTable[iTotalIdxWrite].uiSize	:= LEN(pa_tyXMLTable[iTotalIdxWrite].sValue);

	iTotalIdxWrite	:= iTotalIdxWrite + 1;

	pa_tyXMLTable[iTotalIdxWrite].sTitle	:= 'EN';
	pa_tyXMLTable[iTotalIdxWrite].sValue	:= '';
	pa_tyXMLTable[iTotalIdxWrite].uiSize	:= LEN(pa_tyXMLTable[iTotalIdxWrite].sValue);

	iTotalIdxWrite	:= iTotalIdxWrite + 1;

	iTotalIdxWrite	:= fHermesFormReplyWorkOrderInfo;

END_FUNCTION
```

#### fHermesGenerateBrdAvlDat.st - not listed in the package file held
```iecst
(* Hermes Add One Message Send Buffer *)
FUNCTION fHermesGenerateBrdAvlDat

	fHermesGenerateBrdAvlDat := 0;
	memset(ADR(p_tyHermesBrdAvlDat.a_tyXMLTableDataBrdAvl),0,SIZEOF(p_tyHermesBrdAvlDat.a_tyXMLTableDataBrdAvl));

	pa_usiMacAddr ACCESS tyHermesBAMsgAttribAddr.udiDateTimeForGUID;
	p_tyDTStructure ACCESS tyHermesBAMsgAttribAddr.udiDateTimeForGUID;
	fHermesGenerateUUID(ADR(tyGenBoardAvailable.tyData.sBoardId) , p_tyDTStructure , pa_usiMacAddr);

	memcpy(ADR(tyGenBoardAvailable.tyData.sBoardIdCreatedBy) , tyHermesBAMsgAttribAddr.udiBoardIdCreatedBy  ,SIZEOF(tyGenBoardAvailable.tyData.sBoardIdCreatedBy)) ;
	memcpy(ADR(tyGenBoardAvailable.tyData.sProductTypeId) , tyHermesBAMsgAttribAddr.udiProductTypeId ,SIZEOF(tyGenBoardAvailable.tyData.sProductTypeId)) ;

	p_diWidth ACCESS tyHermesBAMsgAttribAddr.udiWidth;
	diWidthInMM := p_diWidth;
	tyGenBoardAvailable.tyData.rWidth := DINT_TO_REAL(diWidthInMM /1000);

	tyGenBoardAvailable.tyAvl.bBoardId			:= tyGenBoardAvailable.tyData.sBoardId <> '';
	tyGenBoardAvailable.tyAvl.bBoardIdCreatedBy := tyGenBoardAvailable.tyData.sBoardIdCreatedBy <> '';
	tyGenBoardAvailable.tyAvl.bProductTypeId := tyGenBoardAvailable.tyData.sProductTypeId <> '';
	tyGenBoardAvailable.tyAvl.bWidth := tyGenBoardAvailable.tyData.rWidth <> 0;
	tyGenBoardAvailable.tyAvl.bFailedBoard := TRUE;
	tyGenBoardAvailable.tyAvl.bFlippedBoard := TRUE;

	fHermesFormBoardAvailable(ADR(p_tyHermesBrdAvlDat.a_tyXMLTableDataBrdAvl),p_tyDTStructure,tyGenBoardAvailable);
	p_tyHermesBrdAvlDat.iXMLTableDataBrdAvlTtlIdx := 80;
	p_tyHermesBrdAvlDat.bNewBrdAvl := FALSE;

END_FUNCTION
```

#### fHermesSrchAttribValueBrdAvlDat.st - not listed in the package file held
```iecst
(* Hermes Search Attribute Value from BrvAvlDat , return the attribute index value*)
FUNCTION fHermesSrchAttribValueBrdAvlDat

	fHermesSrchAttribValueBrdAvlDat := -1;
	fConvertToLower_254(ADR(sTitleLowerCase) , sAttributeTiltle);
	sAttributeValue := '';

	FOR i := 0 TO 200 DO //search for the board action and update / add if not exist
		IF (p_tyHermesBrdAvlDat.a_tyXMLTableDataBrdAvl[i].sTitle = 'AT') THEN
			fConvertToLower_254(ADR(sLowerCase) , p_tyHermesBrdAvlDat.a_tyXMLTableDataBrdAvl[i].sValue);
			IF (sLowerCase = sTitleLowerCase) THEN
				IF p_tyHermesBrdAvlDat.a_tyXMLTableDataBrdAvl[i+1].sTitle = 'AV' THEN
					sAttributeValue  := p_tyHermesBrdAvlDat.a_tyXMLTableDataBrdAvl[i+1].sValue	; //if Action already in XMLTable
					fHermesSrchAttribValueBrdAvlDat := i;
					EXIT;
				END_IF
			END_IF
		END_IF
	END_FOR

END_FUNCTION
```

- Visualisation Logical/UI/Visu (not shown)

### UI.typ - Do Not Change!!!
```iecst
(*2019-04-04*)
(**)

TYPE
	eUIAction :
		(
		UIActIdle,
		UIActInitial
		);
	eUIInitial :
		(
		UIInitialC0005,
		UIInitialC0007,
		UIInitialP0000,
		UIInitialP0200,
		UIInitialP0201,
		UIInitialP0300,
		UIInitialP0400,
		UIInitialP0900,
		UIInitialP0910,
		UIInitialP0920,
		UIInitialP0922,
		UIInitialP0924,
		UIInitialP0927,
		UIInitialP0928,
		UIInitialP0931,
		UIInitialP0934,
		UIInitialP0935,
		UIInitialP0940,
		UIInitialP1000,
		UIInitialP1020,
		UIInitialP1021,
		UIInitialP1022,
		UIInitialP1023,
		UIInitialP1024,
		UIInitialP1026,
		UIInitialP1040,
		UIInitialP1050,
		UIInitialP1080,
		UIInitialP1081,
		UIInitialDone
		);
END_TYPE

(*Global Alarm*)

TYPE
	tyUIAllAlm : 	STRUCT
		bAlm : ARRAY[0..9999]OF BOOL;
		bWarning : ARRAY[0..9999]OF BOOL;
	END_STRUCT;
END_TYPE
```

### UI.var - Change By Project
```iecst
(*2020-10-08*)
(**)
(*Action & State & Status*)
VAR
	p_UIStat : UDINT;
	p_UIStatus : UDINT;
	p_UIStatTxt : UDINT;
END_VAR
(**)
(*Alarm*)
(**)
(*Output*)
VAR
	p_UIStartupAct : UDINT;
	p_UIHWInfoAct : UDINT;
	p_UITLBuzAct : UDINT;
	p_UIRstErrAct : UDINT;
	p_UIProdRcpAct : UDINT;
	p_UIMpProdRcpAct : UDINT;
	p_UIMcParamAct : UDINT;
	p_UIUsrMgmtAct : UDINT;
	p_UIUSSMEMAAct : UDINT;
	p_UIDSSMEMAAct : UDINT;
	p_UIUSSMEMA2Act : UDINT;
	p_UIStopperAct : UDINT;
	p_UIConvAct : UDINT;
	p_UIAWOpenAct : UDINT;
	p_UIInvertAct : UDINT;
	p_UIOpsAct : UDINT;
	p_UIHermesAct : UDINT;
	p_UILFLeaderAct : UDINT;
	p_UIDOAct : UDINT;
	p_UIClampAct : UDINT;
	p_UIInShutterAct : UDINT;
	p_UIOutShutterAct : UDINT;
	p_UIClamp1Act : UDINT;
	p_UIClamp2Act : UDINT;
	p_UIClamp3Act : UDINT;
END_VAR
(**)
VAR
	p_UIMcParamWr : UDINT;
END_VAR
(**)
VAR
	p_UIProdRcpInfoIn : UDINT;
	p_UIProdRcpSearch : UDINT;
	p_UIProdRcpScan : UDINT;
	p_UIProdRcpCurrRcpWr : UDINT;
END_VAR
(**)
VAR
	p_UIUsrMgmtInfoIn : UDINT;
	p_UIUsrMgmtAccessRightLvl1Wr : UDINT;
	p_UIUsrMgmtAccessRightLvl2Wr : UDINT;
	p_UIUsrMgmtAccessRightLvl3Wr : UDINT;
END_VAR
(**)
VAR
	p_UIHermesUSParamWr : UDINT;
	p_UIHermesDSParamWr : UDINT;
	p_UIHermesSvyParamWr : UDINT;
END_VAR
(**)
VAR
	p_UISetIPAddr : UDINT;
	p_UISetSubnetMask : UDINT;
	p_UINetworkMode : UDINT;
END_VAR
(**)
VAR
	p_UIMnlMod : UDINT;
	p_UIUIMnlMod : UDINT;
	p_UIMuteBuz : UDINT;
END_VAR
(**)
VAR
	p_UIMnlAWGoWidth : UDINT;
	p_UIMnlAWNomSpd : UDINT;
	p_UIMnlAWTargetPos : UDINT;
	p_UIMnlAWStepSize : UDINT;
	p_UIMnlAWJogSpd : UDINT;
END_VAR
(**)
VAR
	p_UIMnlInvertNomSpd : UDINT;
	p_UIMnlInvertTargetPos : UDINT;
	p_UIMnlInvertStepSize : UDINT;
	p_UIMnlInvertJogSpd : UDINT;
END_VAR
(**)
VAR
	p_UIVSMEMAUSEn : UDINT;
	p_UIVSMEMADSEn : UDINT;
	p_UIVSMEMAUBA : UDINT;
	p_UIVSMEMAUBAStat : UDINT;
	p_UIVSMEMADSB : UDINT;
	p_UIVSMEMAUS2En : UDINT;
	p_UIVSMEMAUBA2 : UDINT;
	p_UIVSMEMAUBAStat2 : UDINT;
END_VAR
(**)
VAR
	p_UILeaderRun : UDINT;
END_VAR
(**)
VAR
	p_UIProdAccData : UDINT;
END_VAR
(**)
VAR
	p_UIOpsBypsInitConv : UDINT;
END_VAR
(**)
VAR
	p_UIRlsNewProd : UDINT;
END_VAR
(**)
VAR
	p_UIConvDCCtrl : UDINT;
END_VAR
(**)
VAR
	p_UIInvertDCCtrl : UDINT;
END_VAR
(**)
VAR
	p_UIInvertDCModBrakePress : UDINT;
END_VAR
(**)
VAR
	p_UIMismatchOverWriteConfig : UDINT;
	p_UITempAddrFillDone : UDINT;
	p_UIIPConfigChgDone : UDINT;
	p_UIOverwriteIP : UDINT;
	p_UIOverwriteSubnet : UDINT;
	p_UIOverwriteEthMode : UDINT;
END_VAR
(**)
VAR
	p_UISongTitile : UDINT;
	p_UISongPlay : UDINT;
END_VAR
(*Insert your comment here.*)
VAR
	p_UIBypassTopCover1 : UDINT;
	p_UIMachineSafetySigToDS : UDINT;
	p_UIMachineSafetySigToUS : UDINT;
	p_UISafetyTopCoverSWCoil1 : UDINT;
	p_UITopCvrUnlckToUS : UDINT;
	p_UITopCvrUnlckToDS : UDINT;
	p_UICoverPBLED1 : UDINT;
END_VAR
(**)
VAR
	p_UIMnlModBypassTopCover1 : UDINT;
	p_UIMnlModMachineSafetySigToDS : UDINT;
	p_UIMnlModMachineSafetySigToUS : UDINT;
	p_UIMnlModSafetyTopCoverSWCoil1 : UDINT;
	p_UIMnlModTopCvrUnlckToUS : UDINT;
END_VAR
(**)
VAR
	p_UIMnlModTopCvrUnlckToDS : UDINT;
	p_UIMnlModCoverPBLED1 : UDINT;
END_VAR
(**)
VAR
	p_UIDSTranErr : UDINT;
END_VAR
(**)
VAR
	p_UIRtnBrdReset : UDINT;
	p_UIRtnBrdResetBtn : UDINT;
END_VAR
(**)
VAR
	p_UISimuAct : UDINT;
	p_UIMnlSimu : UDINT;
	P_UISectionLdr : UDINT;
END_VAR
(*Insert your comment here.*)
VAR
	p_UISaveHMIConfigure : UDINT;
	p_UISaveHMISvyConfig : UDINT;
	p_UIQueryBoardInfo : UDINT;
END_VAR
```

### Program Logical/UI/UI (IEC) - 1.00.0 - NtUI v5.00.0 (2018-12-01)

#### Init.st - Change By Project
```iecst
(** 2020-10-06 **)
PROGRAM _INIT

	(* Always Change If Project Change *)

	//Pass Address To Global Address For External Use
	//Action, State & Status
	p_UIStat	:= ADR(eStat);
	p_UIStatus	:= ADR(eStatus);
	p_UIStatTxt	:= ADR(sStatTxt);

	//Alarm

	//Output
	p_UIStartupAct					:= ADR(eStartupAct);
	p_UIHWInfoAct					:= ADR(eHWInfoAct);
	p_UITLBuzAct					:= ADR(eTLBuzAct);
	p_UIRstErrAct					:= ADR(eRstErrAct);
	p_UIProdRcpAct					:= ADR(eProdRcpAct);
	p_UIMpProdRcpAct				:= ADR(eMpProdRcpAct);
	p_UIMcParamAct					:= ADR(eMcParamAct);
	p_UIUsrMgmtAct					:= ADR(eUsrMgmtAct);
	p_UIUSSMEMAAct					:= ADR(eUSSMEMAAct);
	p_UIDSSMEMAAct					:= ADR(eDSSMEMAAct);
	p_UIUSSMEMA2Act					:= ADR(eUSSMEMA2Act);
	p_UIStopperAct					:= ADR(eStopperAct);
	p_UIConvAct						:= ADR(eConvAct);
	p_UIAWOpenAct					:= ADR(eAWOpenAct);
	p_UIInvertAct					:= ADR(eInvertAct);
	p_UIOpsAct						:= ADR(eOpsAct);
	p_UIHermesAct					:= ADR(eHermesAct);
	p_UILFLeaderAct					:= ADR(eLFLeaderAct);
	p_UIDOAct						:= ADR(eDOAct);
	p_UIClampAct					:= ADR(eClampAct);
	p_UIInShutterAct 				:= ADR(eInShutterAct);
	p_UIOutShutterAct 				:= ADR(eOutShutterAct);
	p_UIClamp1Act	 				:= ADR(eClamp1Act);
	p_UIClamp2Act	 				:= ADR(eClamp2Act);
	p_UIClamp3Act	 				:= ADR(eClamp3Act);

	p_UIMcParamWr					:= ADR(tyMcParamWr);

	p_UIProdRcpInfoIn				:= ADR(tyProdRcpInfoIn);
	p_UIProdRcpSearch				:= ADR(sProdRcpSearch);
	p_UIProdRcpScan					:= ADR(sProdRcpScan);
	p_UIProdRcpCurrRcpWr			:= ADR(tyProdRcpCurrRcpWr);

	p_UIUsrMgmtInfoIn				:= ADR(tyUsrMgmtInfoIn);
	p_UIUsrMgmtAccessRightLvl1Wr	:= ADR(tyUsrMgmtAccessRightLvl1Wr);
	p_UIUsrMgmtAccessRightLvl2Wr	:= ADR(tyUsrMgmtAccessRightLvl2Wr);
	p_UIUsrMgmtAccessRightLvl3Wr	:= ADR(tyUsrMgmtAccessRightLvl3Wr);

	p_UIHermesUSParamWr				:= ADR(a_tyHermesUSParamWr);
	p_UIHermesDSParamWr				:= ADR(a_tyHermesDSParamWr);
	p_UIHermesSvyParamWr			:= ADR(tyHermesSvyParamWr);

	p_UISetIPAddr					:= ADR(sSetIPAddr);
	p_UISetSubnetMask				:= ADR(sSetSubnetMask);
	p_UINetworkMode					:= ADR(usiNetworkModeSelected);

	p_UIMnlMod						:= ADR(bManualMod);
	p_UIUIMnlMod					:= ADR(bUIManualMod);
	p_UIMuteBuz						:= ADR(bMuteBuz);

	p_UIMnlAWGoWidth				:= ADR(diMnlAWGoWidth);
	p_UIMnlAWNomSpd					:= ADR(diMnlAWNomSpd);
	p_UIMnlAWTargetPos				:= ADR(diMnlAWTargetPos);
	p_UIMnlAWStepSize				:= ADR(diMnlAWStepSize);
	p_UIMnlAWJogSpd					:= ADR(diMnlAWJogSpd);

	p_UIMnlInvertNomSpd				:= ADR(diMnlInvertNomSpd);
	p_UIMnlInvertTargetPos			:= ADR(diMnlInvertTargetPos);
	p_UIMnlInvertStepSize			:= ADR(diMnlInvertStepSize);
	p_UIMnlInvertJogSpd				:= ADR(diMnlInvertJogSpd);

	p_UIVSMEMAUSEn					:= ADR(bVSMEMAUSEn);
	p_UIVSMEMADSEn					:= ADR(bVSMEMADSEn);
	p_UIVSMEMAUBA					:= ADR(bVSMEMAUBA);
	p_UIVSMEMAUBAStat				:= ADR(bVSMEMAUBAStat);
	p_UIVSMEMADSB					:= ADR(bVSMEMADSB);

	p_UIVSMEMAUS2En					:= ADR(bVSMEMAUS2En);
	p_UIVSMEMAUBA2					:= ADR(bVSMEMAUBA2);
	p_UIVSMEMAUBAStat2				:= ADR(bVSMEMAUBAStat2);

	p_UILeaderRun					:= ADR(bLeaderRun);

	p_UIProdAccData					:= ADR(bProdAccData);

	p_UIOpsBypsInitConv				:= ADR(bOpsBypsInitConv);

	p_UIRlsNewProd					:= ADR(bRlsNewProd);

	p_UIConvDCCtrl					:= ADR(tyP0931ConvInv.tyConvCom.tyBtnDCCtrl.bValue);

	//	p_UIInvertDCCtrl				:= ADR(tyP0931ConvInv.tyInvCom.tyBtnDCCtrl.bValue);

	//	p_UIInvertDCModBrakePress		:= ADR(tyP0931ConvInv.tyInvDC.tyBtnBrake.bValue);

	p_UIMismatchOverWriteConfig		:= ADR(bMismatchOverWriteConfig);
	p_UITempAddrFillDone			:= ADR(bTempAddrFillDone);
	p_UIIPConfigChgDone				:= ADR(bIPConfigChgDone);
	p_UIOverwriteIP					:= ADR(bOverwriteIP);
	p_UIOverwriteSubnet				:= ADR(bOverwriteSubnet);
	p_UIOverwriteEthMode			:= ADR(bOverwriteEthMode);
	(* Always Change If Project Change *)

	p_UISongTitile					:= ADR(uiSongIndex);
	p_UISongPlay					:= ADR(bSongEn);

	// ADD
	p_UIBypassTopCover1				:= ADR(bBypassTopCover1);
	p_UIMachineSafetySigToDS		:= ADR(bMachineSafetySigToDS);
	p_UIMachineSafetySigToUS		:= ADR(bMachineSafetySigToUS);
	p_UISafetyTopCoverSWCoil1		:= ADR(bTopCoverSwitchCoil1);
	p_UITopCvrUnlckToUS				:= ADR(bUnlockCover1Req);
	p_UITopCvrUnlckToDS				:= ADR(bUnlockCover1Req);
	p_UICoverPBLED1					:= ADR(bCoverPBLED1);

	p_UIMnlModBypassTopCover1		:= ADR(bMnlModBypassTopCover1);
	p_UIMnlModMachineSafetySigToDS	:= ADR(bMnlModMachineSafetySigToDS);
	p_UIMnlModMachineSafetySigToUS	:= ADR(bMnlModMachineSafetySigToDS);
	p_UIMnlModSafetyTopCoverSWCoil1	:= ADR(bMnlModTopCoverSwitch1);
	p_UIMnlModTopCvrUnlckToUS		:= ADR(bMnlModUnlockCover1Req);
	p_UIMnlModTopCvrUnlckToDS		:= ADR(bMnlModUnlockCover1Req);
	p_UIMnlModCoverPBLED1			:= ADR(bMnlModCoverPBLED1);

	// ADD
	p_UIDSTranErr 					:= ADR(bDSTranErr);

	//Reset Waiting Return Board
	p_UIRtnBrdReset					:= ADR(bRtnBrdReset);
	p_UIRtnBrdResetBtn				:= ADR(tyP0200OpsGen.tyOps.tyBtnPCBReset.bValue);

	p_UISimuAct						:= ADR(eSimuAct);
	p_UIMnlSimu						:= ADR(bSimuMod);

	P_UISectionLdr					:= ADR(tyP1022McSetVComm.tyLF.tyBtnSectionLdr.bValue);

	p_UISaveHMIConfigure            := ADR(bSaveHMIConfigure);
	p_UISaveHMISvyConfig            := ADR(bSaveHMISvyConfig);
	p_UIQueryBoardInfo				:= ADR(bQueryBoardInfo);
	//p_UITopBarcode                  := ADR(tyP0201OpsConv.tyQueryBoardInfo.tyStringTopBarcode.sValue);
	//p_UIBottomBarcode               := ADR(tyP0201OpsConv.tyQueryBoardInfo.tyStringBottomBarcode.sValue);

END_PROGRAM
```

#### Act_InitGlobal.st - Change By Project
```iecst
(** 2020-10-08 **)
ACTION Act_InitGlobal:

	//Get Data from Global to Internal Use
	p_eAct ACCESS p_StartupUIAct;

	p_bStartupRun ACCESS p_StartupRun;
	p_eStartupStat ACCESS p_StartupStat;
	p_eStartupStatus ACCESS p_StartupStatus;
	p_sStartupStatTxt ACCESS p_StartupStatTxt;
	p_eStartupStep ACCESS p_StartupStep;
	p_sStartupStepTxt ACCESS p_StartupStepTxt;
	p_bStartupGetConfigDone ACCESS p_StartupGetConfigDone;
	p_bStartupMismatchSetConfigDone ACCESS p_StartupMismatchSetConfigDone;
	p_bStartupUISettingsLoadDone ACCESS p_StartupUISettingsLoadDone;

	p_eTLBuzStat ACCESS p_TLBuzStat;
	p_eTLBuzStatus ACCESS p_TLBuzStatus;
	p_sTLBuzStatTxt ACCESS p_TLBuzStatTxt;

	p_tyAlarmCurrList ACCESS p_AlarmCurrList;
	p_tyAlarmRcyList ACCESS p_AlarmRecoveryList;
	p_tyAlarmHistoryList ACCESS p_AlarmHistoryList;
	p_bAlarmWarning ACCESS p_AlarmWarning;
	p_bAlarmErr ACCESS p_AlarmErr;
	p_bAlarmInfo ACCESS p_AlarmInfo;
	p_bAlarmInfoLF ACCESS p_AlarmInfoLF;
	p_sAlarmInfoMsg ACCESS p_AlarmInfoMsg;

	p_eRstErrStat ACCESS p_RstErrStat;
	p_eRstErrStatus ACCESS p_RstErrStatus;
	p_sRstErrStatTxt ACCESS p_RstErrStatTxt;

	p_eHWInfoStat ACCESS p_HWInfoStat;
	p_eHWInfoStatus ACCESS p_HWInfoStatus;
	p_sHWInfoStatTxt ACCESS p_HWInfoStatTxt;
	p_sHWInfoIPAddr ACCESS p_HWInfoIPAddr;
	p_sHWInfoSubnetMask ACCESS p_HWInfoSubnetMask;
	p_udiHWInfoEthMode ACCESS p_HWInfoEthMode;

	p_eProdRcpStat ACCESS p_ProdRcpStat;
	p_eProdRcpStatus ACCESS p_ProdRcpStatus;
	p_sProdRcpStatTxt ACCESS p_ProdRcpStatTxt;
	p_tyProdRcpCurrList	ACCESS p_ProdRcpCurrList;
	p_tyProdRcpFilterList ACCESS p_ProdRcpFilterList;
	p_tyProdRcpSortedList ACCESS p_ProdRcpSortedList;
	p_bProdRcpNmEmpty ACCESS p_ProdRcpNmEmpty;
	p_bProdRcpListFull ACCESS p_ProdRcpListFull;
	p_bProdRcpNmNotExist ACCESS p_ProdRcpNmNotExist;
	p_tyProdRcpInfoOut ACCESS p_ProdRcpInfoOut;
	p_tyProdRcpCurrRcp0 ACCESS p_ProdRcpCurrRcp0;
	p_tyProdRcpCurrRcp1 ACCESS p_ProdRcpCurrRcp1;
	p_tyProdRcpCurrRcp2 ACCESS p_ProdRcpCurrRcp2;

	p_eMpProdRcpStat ACCESS p_MpProdRcpStat;
	p_eMpProdRcpStatus ACCESS p_MpProdRcpStatus;

	p_eMcParamStat ACCESS p_McParamStat;
	p_eMcParamStatus ACCESS p_McParamStatus;
	p_sMcParamStatTxt ACCESS p_McParamStatTxt;
	p_tyMcParamCurr	ACCESS p_McParamCurr;

	p_tyNtParamCurr ACCESS p_NtParamCurr;

	p_eUsrMgmtStat ACCESS p_UsrMgmtStat;
	p_eUsrMgmtStatus ACCESS p_UsrMgmtStatus;
	p_sUsrMgmtStatTxt ACCESS p_UsrMgmtStatTxt;
	p_tyUsrMgmtCurrUsr ACCESS p_UsrMgmtCurrUsr;
	p_tyUsrMgmtCurrAccessRgt ACCESS p_UsrMgmtCurrAccessRight;
	p_tyUsrMgmtAllList ACCESS p_UsrMgmtAllList;
	p_tyUsrMgmtLv2List ACCESS p_UsrMgmtLvl2List;
	p_tyUsrMgmtLv3List ACCESS p_UsrMgmtLvl3List;
	p_tyUsrMgmtAdminList ACCESS p_UsrMgmtAdminList;
	p_bUsrMgmtNmEmpty ACCESS p_UsrMgmtNmEmpty;
	p_bUsrMgmtListFull ACCESS p_UsrMgmtListFull;
	p_bUsrMgmtNmExist ACCESS p_UsrMgmtNmExist;
	p_bUsrMgmtNmNotExist ACCESS p_UsrMgmtNmNotExist;
	p_bUsrMgmtLastAdmin ACCESS p_UsrMgmtLastAdmin;
	p_bUsrMgmtLoginSuccess ACCESS p_UsrMgmtLoginSuccess;
	p_bUsrMgmtPwMismatch ACCESS p_UsrMgmtPwMismatch;
	p_bUsrMgmtUnableDelete ACCESS p_UsrMgmtUnableDelete;
	p_tyUsrMgmtFullData ACCESS p_UsrMgmtFullData;

	p_eUSSMEMAStat ACCESS p_USSMEMAStat;
	p_eUSSMEMAStatus ACCESS p_USSMEMAStatus;
	p_sUSSMEMAStatTxt ACCESS p_USSMEMAStatTxt;
	p_bUSSMEMAUSRdy ACCESS p_USSMEMAUSRdy;
	p_bUSSMEMAUSGdBrdRdy ACCESS p_USSMEMAUSGdBrdRdy;
	p_bUSSMEMADSRdy ACCESS p_USSMEMADSRdy;
	p_bUSSMEMAUSB ACCESS p_USSMEMAUSB;

	p_eDSSMEMAStat ACCESS p_DSSMEMAStat;
	p_eDSSMEMAStatus ACCESS p_DSSMEMAStatus;
	p_sDSSMEMAStatTxt ACCESS p_DSSMEMAStatTxt;
	p_bDSSMEMAUSRdy ACCESS p_DSSMEMAUSRdy;
	p_bDSSMEMAUSGdBrdRdy ACCESS p_DSSMEMAUSGdBrdRdy;
	p_bDSSMEMADSRdy	ACCESS p_DSSMEMADSRdy;
	p_bDSSMEMADBA ACCESS p_DSSMEMADBA;
	p_bDSSMEMADBAStat ACCESS p_DSSMEMADBAStat;

	//UpStreamSMEMA2
	p_eUSSMEMA2Stat ACCESS p_USSMEMA2Stat;
	p_eUSSMEMA2Status ACCESS p_USSMEMA2Status;
	p_sUSSMEMA2StatTxt ACCESS p_USSMEMA2StatTxt;
	p_bUSSMEMA2USRdy ACCESS p_USSMEMA2USRdy;
	p_bUSSMEMA2USGdBrdRdy ACCESS p_USSMEMA2USGdBrdRdy;
	p_bUSSMEMA2DSRdy ACCESS p_USSMEMA2DSRdy;
	p_bUSSMEMA2USB ACCESS p_USSMEMA2USB;
	p_bUSSMEMA2Transporting ACCESS p_USSMEMA2Transporting;

	p_bUSHermesUSRdy ACCESS p_USHermesUSRdy;
	p_bUSHermesDSRdy ACCESS p_USHermesDSRdy;
	p_bUSHermesUSGdRdy ACCESS p_USHermesUSGdRdy;
	p_bUSHermesDSGdRdy ACCESS p_USHermesDSGdRdy;
	p_bUSHermesConnected ACCESS p_USHermesConnected;
	p_bUSHermesAccDataMnl ACCESS p_USHermesAccDataMnl;

	p_bDSHermesUSRdy ACCESS p_DSHermesUSRdy;
	p_bDSHermesDSRdy ACCESS p_DSHermesDSRdy;
	p_bDSHermesUSGdRdy ACCESS p_DSHermesUSGdRdy;
	p_bDSHermesDSGdRdy ACCESS p_DSHermesDSGdRdy;
	p_bDSHermesConnected ACCESS p_DSHermesConnected;

	p_eConvStat ACCESS p_ConvStat;
	p_eConvStatus ACCESS p_ConvStatus;
	p_sConvStatTxt ACCESS p_ConvStatTxt;

	p_bConvHvBrd ACCESS p_OpsInvertHvBrd;
	p_bConvGdBrd ACCESS p_OpsInvertGdBrd;

	p_eAWOpenStat ACCESS p_AWOpenStat;
	p_eAWOpenStatus ACCESS p_AWOpenStatus;
	p_sAWOpenStatTxt ACCESS p_AWOpenStatTxt;
	p_udiAWOpenAxisErrID ACCESS p_AWOpenAxisErrID;
	p_bAWOpenAxisErr ACCESS p_AWOpenAxisErr;
	p_bAWOpenPwrOn ACCESS p_AWOpenPwrOn;
	p_bAWOpenIsHomed ACCESS p_AWOpenIsHomed;
	p_diAWOpenActualPos ACCESS p_AWOpenActualPos;
	p_bAWOpenFwdLmtSen ACCESS p_AWOpenFwdLmtSen;
	p_bAWOpenRevLmtSen ACCESS p_AWOpenRevLmtSen;
	p_sAWOpenAxisErrTxt ACCESS p_AWOpenAxisErrTxt;
	p_bAWOpenJogging ACCESS p_AWOpenJogging;
	p_bAWOpenOpenSen ACCESS p_AWOpenOpenSen;
	p_bAWOpenCloseSen ACCESS p_AWOpenCloseSen;

	p_eInvertStat ACCESS p_MotorBrkStat;
	p_eInvertStatus ACCESS p_MotorBrkStatus;
	p_sInvertStatTxt ACCESS p_MotorBrkStatTxt;

	p_eOpsStat ACCESS p_OpsStat;
	p_eOpsStatus ACCESS p_OpsStatus;
	p_sOpsStatTxt ACCESS p_OpsStatTxt;
	p_eOpsOpsStatus ACCESS p_OpsOpsStatus;

	p_sOpsInvertStepTxt ACCESS p_OpsInvertStepTxt;
	p_eOpsInvertCurrPos ACCESS p_OpsInvertInvertCurrPos;

	p_bOpsInvertStepInitConv ACCESS p_OpsInvertStepInitConv;
	p_bOpsInvertStepInitDone ACCESS p_OpsInvertStepInitDone;

	p_bOpsStatusRun ACCESS p_OpsStatusRun;
	p_bOpsStatusStop ACCESS p_OpsStatusStop;
	p_bOpsStatusCycleStop ACCESS p_OpsStatusCycleStop;
	p_bOpsStatusStep ACCESS p_OpsStatusStep;
	p_bOpsRun ACCESS p_OpsRun;

	p_bOpsUSStandby ACCESS p_OpsInvertStepUSStandby;
	p_bOpsDSStandby ACCESS p_OpsInvertStepDSStandby;

	// ADD safetySignal
	p_bOpsInvertStepAWMove ACCESS p_OpsInvertStepAWMove;
	p_bOpsSafeMode ACCESS p_OpsInvertStepOpsSafeMode;

	p_eHermesStat ACCESS p_HermesStat;
	p_eHermesStatus ACCESS p_HermesStatus;
	p_tyHermesConfiguration ACCESS p_HermesConfiguration;

	p_eLFLeaderStat ACCESS p_LFLeaderStat;
	p_eLFLeaderStatus ACCESS p_LFLeaderStatus;
	p_tyLFLeaderFollowerInfo ACCESS p_LFLeaderFollowerInfo;
	p_tyLFLeaderFollowerToLeaderTag ACCESS p_LFLeaderFollowerToLeaderTag;

	p_bLFFollowerProdAccDataMnl ACCESS p_LFFollowerProdAccDataMnl;
	p_bLFFollowerLdrSeqCtrlInActive ACCESS p_LFFollowerLdrSeqCtrlInActive;
	p_bLFFollowerUSAllow ACCESS p_LFFollowerUSAllow;
	p_bLFFollowerDSAllow ACCESS p_LFFollowerDSAllow;

	p_bFollower1WaitRlsProd ACCESS p_Follower1WaitRlsBrd;

	p_bLCSLFAccDataMnl ACCESS p_LCSLFAccDataMnl;

	p_tyDI ACCESS p_DI;

	p_tyDO ACCESS p_DO;
	p_eDOStat ACCESS p_DOStat;
	p_eDOStatus ACCESS p_DOStatus;

	//Stopper
	p_eStopperStat ACCESS p_PneuNoSenStopperStat;
	p_eStopperStatus ACCESS p_PneuNoSenStopperStatus;
	p_sStopperStatTxt ACCESS p_PneuNoSenStopperStatTxt;
	p_bStopperTwoCtrlOut ACCESS p_PneuNoSenStopperTwoCtrlOut;
	p_bStopperExtCtrl ACCESS p_PneuNoSenStopperExtCtrl;
	p_bStopperRetCtrl ACCESS p_PneuNoSenStopperRetCtrl;
	p_bStopperExtended ACCESS p_PneuNoSenStopperExtended;

	//Clamp
	p_eClampStat ACCESS p_PneuNoSenClampStat;
	p_eClampStatus ACCESS p_PneuNoSenClampStatus;
	p_sClampStatTxt ACCESS p_PneuNoSenClampStatTxt;
	p_bClampTwoCtrlOut ACCESS p_PneuNoSenClampTwoCtrlOut;
	p_bClampExtCtrl ACCESS p_PneuNoSenClampExtCtrl;
	p_bClampRetCtrl ACCESS p_PneuNoSenClampRetCtrl;

	//Shutter
	p_eInShutterStat ACCESS p_Pneu2SenInShutterStat;
	p_eInShutterStatus ACCESS p_Pneu2SenInShutterStatus;
	p_sInShutterStatTxt ACCESS p_Pneu2SenInShutterStatTxt;
	p_bInShutterExtCtrl ACCESS p_Pneu2SenInShutterExtCtrl;
	p_bInShutterRetCtrl ACCESS p_Pneu2SenInShutterRetCtrl;
	p_bInShutterTwoCtrlOut ACCESS p_Pneu2SenInShutterTwoCtrlOut;
	p_bInShutterExtended ACCESS p_Pneu2SenInShutterExtended;
	p_bInShutterRetracted ACCESS p_Pneu2SenInShutterRetracted;

	p_eOutShutterStat ACCESS p_Pneu2SenOutShutterStat;
	p_eOutShutterStatus ACCESS p_Pneu2SenOutShutterStatus;
	p_sOutShutterStatTxt ACCESS p_Pneu2SenOutShutterStatTxt;
	p_bOutShutterExtCtrl ACCESS p_Pneu2SenOutShutterExtCtrl;
	p_bOutShutterRetCtrl ACCESS p_Pneu2SenOutShutterRetCtrl;
	p_bOutShutterTwoCtrlOut ACCESS p_Pneu2SenOutShutterTwoCtrlOut;
	p_bOutShutterExtended ACCESS p_Pneu2SenOutShutterExtended;
	p_bOutShutterRetracted ACCESS p_Pneu2SenOutShutterRetracted;

	//Clamp1
	p_eClamp1Stat ACCESS p_Pneu2SenClamp1Stat;
	p_eClamp1Status ACCESS p_Pneu2SenClamp1Status;
	p_sClamp1StatTxt ACCESS p_Pneu2SenClamp1StatTxt;
	p_bClamp1ExtCtrl ACCESS p_Pneu2SenClamp1ExtCtrl;
	p_bClamp1RetCtrl ACCESS p_Pneu2SenClamp1RetCtrl;
	p_bClamp1TwoCtrlOut ACCESS p_Pneu2SenClamp1TwoCtrlOut;
	p_bClamp1Extended ACCESS p_Pneu2SenClamp1Extended;
	p_bClamp1Retracted ACCESS p_Pneu2SenClamp1Retracted;

	//Clamp2
	p_eClamp2Stat ACCESS p_Pneu2SenClamp2Stat;
	p_eClamp2Status ACCESS p_Pneu2SenClamp2Status;
	p_sClamp2StatTxt ACCESS p_Pneu2SenClamp2StatTxt;
	p_bClamp2ExtCtrl ACCESS p_Pneu2SenClamp2ExtCtrl;
	p_bClamp2RetCtrl ACCESS p_Pneu2SenClamp2RetCtrl;
	p_bClamp2TwoCtrlOut ACCESS p_Pneu2SenClamp2TwoCtrlOut;
	p_bClamp2Extended ACCESS p_Pneu2SenClamp2Extended;
	p_bClamp2Retracted ACCESS p_Pneu2SenClamp2Retracted;

	//Clamp3
	p_eClamp3Stat ACCESS p_Pneu2SenClamp3Stat;
	p_eClamp3Status ACCESS p_Pneu2SenClamp3Status;
	p_sClamp3StatTxt ACCESS p_Pneu2SenClamp3StatTxt;
	p_bClamp3ExtCtrl ACCESS p_Pneu2SenClamp3ExtCtrl;
	p_bClamp3RetCtrl ACCESS p_Pneu2SenClamp3RetCtrl;
	p_bClamp3TwoCtrlOut ACCESS p_Pneu2SenClamp3TwoCtrlOut;
	p_bClamp3Extended ACCESS p_Pneu2SenClamp3Extended;
	p_bClamp3Retracted ACCESS p_Pneu2SenClamp3Retracted;

	p_bMtrBrkRls ACCESS p_MotorBrkMtrBrkRls;

	p_bLeftSen ACCESS p_DIConvLftSen;
	p_bRightSen	ACCESS p_DIConvRgtSen;
	p_diInitTm ACCESS p_McParamConvInitTm;
	p_eDirection ACCESS p_NtParamProjConvDir;

	p_bDSSMEMAAlmData ACCESS p_DSSMEMAAlmData;
	p_bConvAlmData ACCESS p_ConvAlmData;

	p_bUnlockCovPrep ACCESS p_NTParamUnlockCovPrep;
	p_bMachineSafetyPrep ACCESS p_NTParamMachineSafetySig;

	p_bOpsInvOnceTwicePCBOut ACCESS p_OpsInvertOnceTwicePCBOut;
	p_bOpsInvertStepUSStandby ACCESS p_OpsInvertStepUSStandby;

	//Simulation
	p_eSimuStat ACCESS p_SimuStat;
	p_eSimuStatus ACCESS p_SimuStatus;

	p_eSimuSimuStatus ACCESS p_SimuSimuStatus;
	p_bSimuStatusRun ACCESS p_SimuStatusRun;
	p_bSimuStatusStop ACCESS p_SimuStatusStop;
	p_bSimuStatusCycleStop ACCESS p_SimuStatusCycleStop;
	p_bSimuStatusStep ACCESS p_SimuStatusStep;

END_ACTION
```

#### Cyclic.st - Do Not Change!!!
```iecst
(** 2019-03-29 **)
PROGRAM _CYCLIC

	IF bInitDone = FALSE THEN
		bInitDone	:= TRUE;

		Act_InitLocal;
		Act_InitGlobal;

	ELSIF bInitialDone = FALSE THEN
		bInitialDone	:= TRUE;

		Act_Initial;

	ELSE

		Act_LinkAction;
		Act_Action;
		Act_Main;
		Act_Background;

	END_IF

END_PROGRAM
```

#### Act_InitLocal.st - Do Not Change!!!
```iecst
(** 2019-03-25 **)
ACTION Act_InitLocal:

	//Input Reference Link To Local Variable
	p_eAct ACCESS ADR(eAct);

END_ACTION
```

#### Act_Initial.st - Change By Project
```iecst
(** 2019-01-03 **)
ACTION Act_Initial:

	//Initial
	sStatTxt	:= a_sStatText[eStat];

END_ACTION
```

#### Act_Action.st - Do Not Change!!!
```iecst
(** 2019-03-25 **)
ACTION Act_Action:

	//Reset Done
	IF eStatus = Done AND p_eAct = UIActIdle THEN
		eStat	:= UIActIdle;
	END_IF

	//Set p_eAct
	IF eStatus = Idle THEN
		eStat	:= p_eAct;
	END_IF

END_ACTION
```

#### Act_Main.st - Do Not Change!!!
```iecst
(** 2019-04-04 **)
ACTION Act_Main:

	//Main
	CASE eStat OF

		UIActIdle:
			IF eStatus <> Idle THEN	//Reset Data
				//Private

				sStatTxt	:= a_sStatText[eStat];

				eUIInit	:= UIInitialC0005;
			END_IF

			eStatus	:= Idle;

		UIActInitial:
			IF eStatus = Idle OR eStatus = Busy THEN

				eStatus	:= Busy;

				sStatTxt	:= a_sStatText[eStat];

				CASE eUIInit OF
					UIInitialC0005:
						Act_Main_C0005;
						eUIInit	 		:= UIInitialC0007;

					UIInitialC0007:
						Act_Main_C0007;
						eUIInit	 		:= UIInitialP0000;

					UIInitialP0000:
						Act_Main_P0000;
						eUIInit	 		:= UIInitialP0200;

					UIInitialP0200:
						Act_Main_P0200;
						eUIInit	 		:= UIInitialP0201;

					UIInitialP0201:
						Act_Main_P0201;
						eUIInit	 		:= UIInitialP0300;

					UIInitialP0300:
						Act_Main_P0300;
						eUIInit	 		:= UIInitialP0400;

					UIInitialP0400:
						Act_Main_P0400;
						eUIInit		 	:= UIInitialP0900;

					UIInitialP0900:
						Act_Main_P0900;
						eUIInit		 	:= UIInitialP0910;

					UIInitialP0910:
						Act_Main_P0910;
						eUIInit		 	:= UIInitialP0920;

					UIInitialP0920:
						Act_Main_P0920;
						eUIInit		 	:= UIInitialP0922;

					UIInitialP0922:
						Act_Main_P0922;
						eUIInit		 	:= UIInitialP0931;

					UIInitialP0931:
						Act_Main_P0931;
						eUIInit		 	:= UIInitialP0934;

					UIInitialP0934:
						Act_Main_P0934;
						eUIInit		 	:= UIInitialP0940;

					UIInitialP0940:
						Act_Main_P0940;
						eUIInit		 	:= UIInitialP1000;

					UIInitialP1000:
						Act_Main_P1000;
						eUIInit		 	:= UIInitialP1020;

					UIInitialP1020:
						Act_Main_P1020;
						eUIInit		 	:= UIInitialP1021;

					UIInitialP1021:
						Act_Main_P1021;
						eUIInit		 	:= UIInitialP1022;

					UIInitialP1022:
						Act_Main_P1022;
						eUIInit		 	:= UIInitialP1023;

					UIInitialP1023:
						Act_Main_P1023;
						eUIInit		 	:= UIInitialP1024;

					UIInitialP1024:
						Act_Main_P1024;
						eUIInit			:= UIInitialP1040;

					UIInitialP1040:
						Act_Main_P1040;
						eUIInit		 	:= UIInitialP1050;

					UIInitialP1050:
						Act_Main_P1050;
						eUIInit		 	:= UIInitialP1080;

					UIInitialP1080:
						Act_Main_P1080;
						eUIInit		 	:= UIInitialP1081;

					UIInitialP1081:
						Act_Main_P1081;
						eUIInit		 	:= UIInitialDone;

					UIInitialDone:
						tyMcParamWr					:= p_tyMcParamCurr;

						tyProdRcpCurrRcpWr			:= p_tyProdRcpCurrRcp0;

						tyUsrMgmtAccessRightLvl1Wr	:= p_tyUsrMgmtFullData.tyAccessRightLvl1;
						tyUsrMgmtAccessRightLvl2Wr	:= p_tyUsrMgmtFullData.tyAccessRightLvl2;
						tyUsrMgmtAccessRightLvl3Wr	:= p_tyUsrMgmtFullData.tyAccessRightLvl3;

						a_tyHermesUSParamWr			:= p_tyHermesConfiguration.a_tyUSParam;
						a_tyHermesDSParamWr			:= p_tyHermesConfiguration.a_tyDSParam;

						eStatus	:= Done;

				END_CASE

			END_IF

	END_CASE

END_ACTION
```

#### Package Logical/UI/UI/Act_Main - Change By Project

#### Act_Main_C0005.st
```iecst
(** 2018-12-21 **)
ACTION Act_Main_C0005:

//	tyCommon.tyMain.tyBtnMuteBuz.uiRtStat.0	:= p_tyNtParamCurr.tyDOSettings.diBuz = 0;

	IF p_tyNtParamCurr.tyDOSettings.diBuz = 0 THEN
		fUIInRtStatHide(ADR(tyCommon.tyMain.tyBtnMuteBuz.uiRtStat));
	ELSE
		fUIInRtStatOff(ADR(tyCommon.tyMain.tyBtnMuteBuz.uiRtStat));
	END_IF

//	fUIInRtStatHide(ADR(tyCommon.tyMain.tyHotspotNaviStart.uiRtStat));
	fUIInRtStatHide(ADR(tyCommon.tyMain.tyBtnAlarm.uiRtStat));

END_ACTION
```

#### Act_Main_C0007.st
```iecst
(** 2018-12-21 **)
ACTION Act_Main_C0007:

	IF p_tyNtParamCurr.bLeaderMc = TRUE THEN
		tyCommon.tyNotif.tyTxtLFMc.usiValueIdx	:= 0;
	ELSE
		tyCommon.tyNotif.tyTxtLFMc.usiValueIdx	:= 1;
	END_IF

END_ACTION
```

#### Act_Main_P0000.st
```iecst
(** 2018-12-21 **)
ACTION Act_Main_P0000:

	//Screen Saver
	tyProperty.tyVisu.uiSSaverTm	:= p_tyMcParamCurr.uiSSaverTmInSec;

END_ACTION
```

#### Act_Main_P0200.st
```iecst
(** 2018-12-21 **)
ACTION Act_Main_P0200:

	//Direction
	CASE p_tyNtParamCurr.eProjConvDir OF
		ConvDirLToR:
			tyP0200OpsGen.tyOps.tyBitmapDir1.usiValueIdx	:= 0;	// -->>
			tyP0200OpsGen.tyOps.tyBitmapDir2.usiValueIdx	:= 0;	// -->>
		ConvDirRToL:
			tyP0200OpsGen.tyOps.tyBitmapDir1.usiValueIdx	:= 1;	// <<--
			tyP0200OpsGen.tyOps.tyBitmapDir2.usiValueIdx	:= 1;	// <<--
		ConvDirLToL:
			tyP0200OpsGen.tyOps.tyBitmapDir1.usiValueIdx	:= 0;	// -->>
			tyP0200OpsGen.tyOps.tyBitmapDir2.usiValueIdx	:= 1;	// <<--
		ConvDirRToR:
			tyP0200OpsGen.tyOps.tyBitmapDir2.usiValueIdx	:= 1;	// <<--
			tyP0200OpsGen.tyOps.tyBitmapDir1.usiValueIdx	:= 0;	// -->>
	END_CASE

	IF p_tyNtParamCurr.tyDOSettings.diTLGreen<>0 OR p_tyNtParamCurr.tyDOSettings.diTLAmber<>0 OR p_tyNtParamCurr.tyDOSettings.diTLRed<>0 THEN
		IF p_tyNtParamCurr.eTLBuzMode=TLBuzModBHTC THEN
			tyP0200OpsGen.tyOps.tyBitmapMc.usiValueIdx := 200;
		ELSE
			tyP0200OpsGen.tyOps.tyBitmapMc.usiValueIdx := 100;
		END_IF
	ELSE
		tyP0200OpsGen.tyOps.tyBitmapMc.usiValueIdx := 0;
	END_IF

	//Hide Warning Bitmap for LF
	fUIInRtStatHide(ADR(tyP0200OpsGen.tyOps.tyTxtLdrInActiveCtrl.uiRtStat));
	fUIInRtStatHide(ADR(tyP0201OpsConv.tyOps.tyTxtLdrInActiveCtrl.uiRtStat));
	fUIInRtStatHide(ADR(tyP0200OpsGen.tyOps.tyBitmapWarningLF.uiRtStat));
	fUIInRtStatHide(ADR(tyP0201OpsConv.tyOps.tyBitmapWarningLF.uiRtStat));

	tyP0200OpsGen.tyOps.tyBtnBypassTopCover1.uiRtStat.0 	:= NOT(p_tyNtParamCurr.bUnlockCoverPrep);

	IF NOT(p_tyNtParamCurr.bProjInvertOncePrep AND p_tyNtParamCurr.bProjInvertTwicePrep) THEN

		fUIInRtStatHide(ADR(tyP0200OpsGen.tyOps.tyTxtUS2.uiRtStat));
		fUIInRtStatHide(ADR(tyP0200OpsGen.tyOps.tyBitmapUSCommIcon2.uiRtStat));
		fUIInRtStatHide(ADR(tyP0200OpsGen.tyOps.tyBitmapUSCommIn2.uiRtStat));
		fUIInRtStatHide(ADR(tyP0200OpsGen.tyOps.tyBitmapUSCommOut2.uiRtStat));
		fUIInRtStatHide(ADR(tyP0200OpsGen.tyOps.tyHotspotUSVirtual2.uiRtStat));
		fUIInRtStatHide(ADR(tyP0200OpsGen.tyUSVSMEMA2.tyLyr.uiRtStat));
		fUIInRtStatHide(ADR(tyP0200OpsGen.tyOps.tyBtnPCBReset.uiRtStat));

	END_IF

END_ACTION
```
